LIN {X 0,Y 253.722,Z 799.815,A -85,B 0,C 180,E1 18671.44,E2 18671.44} C_VEL
LIN {X 0,Y 268.421,Z 770.688,A -85,B 0,C 180,E1 18677.162,E2 18677.162} C_VEL
LIN {X 0,Y 281.731,Z 738.919,A -85,B 0,C 180,E1 18681.257,E2 18681.257} C_VEL
LIN {X 0,Y 284.612,Z 730.237,A -85,B 0,C 180,E1 18682.199,E2 18682.199} C_VEL
LIN {X 0,Y 279.923,Z 708.728,A -85,B 0,C 180,E1 18687.264,E2 18687.264} C_VEL
LIN {X 0,Y 272.289,Z 686.779,A -85,B 0,C 180,E1 18693.595,E2 18693.595} C_VEL
LIN {X 0,Y 264.119,Z 669.28,A -85,B 0,C 180,E1 18700.544,E2 18700.544} C_VEL
LIN {X 0,Y 257.422,Z 656.995,A -85,B 0,C 180,E1 18708.127,E2 18708.127} C_VEL
LIN {X 0,Y 254.132,Z 650.458,A -85,B 0,C 180,E1 18714.879,E2 18714.879} C_VEL
LIN {X 0,Y 253.888,Z 650.396,A -85,B 0,C 180,E1 18725.138,E2 18725.138} C_VEL
LIN {X 0,Y 254.562,Z 652.061,A -85,B 0,C 180,E1 18727.374,E2 18727.374} C_VEL
LIN {X 0,Y 257.625,Z 657.599,A -85,B 0,C 180,E1 18733,E2 18733} C_VEL
LIN {X 0,Y 260.37,Z 676.439,A -85,B 0,C 180,E1 18739.556,E2 18739.556} C_VEL
LIN {X 0,Y 277.56,Z 705.99,A -85,B 0,C 180,E1 18753.063,E2 18753.063} C_VEL
LIN {X 0,Y 289.539,Z 719.07,A -85,B 0,C 180,E1 18759.84,E2 18759.84} C_VEL
LIN {X 0,Y 300.678,Z 730.907,A -85,B 0,C 180,E1 18766.755,E2 18766.755} C_VEL
LIN {X 0,Y 310.062,Z 741.061,A -85,B 0,C 180,E1 18773.393,E2 18773.393} C_VEL
LIN {X 0,Y 317.477,Z 748.305,A -85,B 0,C 180,E1 18779.146,E2 18779.146} C_VEL
LIN {X 0,Y 324.187,Z 754.391,A -85,B 0,C 180,E1 18785.145,E2 18785.145} C_VEL
LIN {X 0,Y 329.073,Z 760.266,A -85,B 0,C 180,E1 18791.212,E2 18791.212} C_VEL
LIN {X 0,Y 333.307,Z 763.024,A -85,B 0,C 180,E1 18796.872,E2 18796.872} C_VEL
LIN {X 0,Y 336.362,Z 764.049,A -85,B 0,C 180,E1 18802.239,E2 18802.239} C_VEL
LIN {X 0,Y 337.345,Z 765.358,A -85,B 0,C 180,E1 18807.428,E2 18807.428} C_VEL
LIN {X 0,Y 337.291,Z 765.495,A -85,B 0,C 180,E1 18812.573,E2 18812.573} C_VEL
LIN {X 0,Y 336.316,Z 764.064,A -85,B 0,C 180,E1 18817.923,E2 18817.923} C_VEL
LIN {X 0,Y 333.217,Z 763.056,A -85,B 0,C 180,E1 18823.132,E2 18823.132} C_VEL
LIN {X 0,Y 329.143,Z 760.264,A -85,B 0,C 180,E1 18828.784,E2 18828.784} C_VEL
LIN {X 0,Y 324.257,Z 754.4,A -85,B 0,C 180,E1 18834.85,E2 18834.85} C_VEL
LIN {X 0,Y 317.504,Z 748.261,A -85,B 0,C 180,E1 18840.862,E2 18840.862} C_VEL
LIN {X 0,Y 309.323,Z 739.929,A -85,B 0,C 180,E1 18847.257,E2 18847.257} C_VEL
LIN {X 0,Y 299.888,Z 729.733,A -85,B 0,C 180,E1 18853.843,E2 18853.843} C_VEL
LIN {X 0,Y 288.152,Z 717.936,A -85,B 0,C 180,E1 18860.906,E2 18860.906} C_VEL
LIN {X 0,Y 276.213,Z 704.369,A -85,B 0,C 180,E1 18867.689,E2 18867.689} C_VEL
LIN {X 0,Y 258.025,Z 670.823,A -85,B 0,C 180,E1 18883.393,E2 18883.393} C_VEL
LIN {X 0,Y 254.267,Z 663.867,A -85,B 0,C 180,E1 18888.836,E2 18888.836} C_VEL
LIN {X 0,Y 252.197,Z 658.099,A -85,B 0,C 180,E1 18894.827,E2 18894.827} C_VEL
LIN {X 0,Y 252.201,Z 658.014,A -85,B 0,C 180,E1 18904.297,E2 18904.297} C_VEL
LIN {X 0,Y 252.963,Z 660.074,A -85,B 0,C 180,E1 18906.977,E2 18906.977} C_VEL
LIN {X 0,Y 256.034,Z 666.467,A -85,B 0,C 180,E1 18912.914,E2 18912.914} C_VEL
LIN {X 0,Y 260.849,Z 675.753,A -85,B 0,C 180,E1 18918.61,E2 18918.61} C_VEL
LIN {X 0,Y 267.694,Z 691.294,A -85,B 0,C 180,E1 18925.184,E2 18925.184} C_VEL
LIN {X 0,Y 274.436,Z 712.152,A -85,B 0,C 180,E1 18931.6,E2 18931.6} C_VEL
LIN {X 0,Y 278.679,Z 732.602,A -85,B 0,C 180,E1 18936.691,E2 18936.691} C_VEL
LIN {X 0,Y 271.431,Z 751.922,A -85,B 0,C 180,E1 18938.973,E2 18938.973} C_VEL
LIN {X 0,Y 257.684,Z 781.058,A -85,B 0,C 180,E1 18943.356,E2 18943.356} C_VEL
LIN {X 0,Y 242.695,Z 808.411,A -85,B 0,C 180,E1 18949.666,E2 18949.666} C_VEL
LIN {X 0,Y 230.265,Z 829.686,A -85,B 0,C 180,E1 18957.149,E2 18957.149} C_VEL
LIN {X 0,Y 221.341,Z 845.658,A -85,B 0,C 180,E1 18965.769,E2 18965.769} C_VEL
LIN {X 0,Y 217.04,Z 855.186,A -85,B 0,C 180,E1 18973.797,E2 18973.797} C_VEL
LIN {X 0,Y 215.382,Z 860.762,A -85,B 0,C 180,E1 18981.918,E2 18981.918} C_VEL
LIN {X 0,Y 215.327,Z 862.605,A -85,B 0,C 180,E1 18990,E2 18990} C_VEL
LIN {X 0,Y 215.382,Z 860.762,A -85,B 0,C 180,E1 18998.082,E2 18998.082} C_VEL
LIN {X 0,Y 217.443,Z 854.155,A -85,B 0,C 180,E1 19007.213,E2 19007.213} C_VEL
LIN {X 0,Y 223.848,Z 841.066,A -85,B 0,C 180,E1 19017.165,E2 19017.165} C_VEL
LIN {X 0,Y 234.929,Z 821.817,A -85,B 0,C 180,E1 19025.991,E2 19025.991} C_VEL
LIN {X 0,Y 247.875,Z 799.283,A -85,B 0,C 180,E1 19032.747,E2 19032.747} C_VEL
LIN {X 0,Y 263.025,Z 770.451,A -85,B 0,C 180,E1 19038.445,E2 19038.445} C_VEL
LIN {X 0,Y 276.907,Z 738.464,A -85,B 0,C 180,E1 19042.564,E2 19042.564} C_VEL
LIN {X 0,Y 278.662,Z 732.639,A -85,B 0,C 180,E1 19043.306,E2 19043.306} C_VEL
LIN {X 0,Y 274.032,Z 710.65,A -85,B 0,C 180,E1 19048.811,E2 19048.811} C_VEL
LIN {X 0,Y 267.257,Z 690.159,A -85,B 0,C 180,E1 19055.22,E2 19055.22} C_VEL
LIN {X 0,Y 260.328,Z 674.883,A -85,B 0,C 180,E1 19061.9,E2 19061.9} C_VEL
LIN {X 0,Y 255.049,Z 664.367,A -85,B 0,C 180,E1 19068.666,E2 19068.666} C_VEL
LIN {X 0,Y 252.498,Z 658.186,A -85,B 0,C 180,E1 19074.846,E2 19074.846} C_VEL
LIN {X 0,Y 252.193,Z 658.115,A -85,B 0,C 180,E1 19085.173,E2 19085.173} C_VEL
LIN {X 0,Y 252.886,Z 661.098,A -85,B 0,C 180,E1 19088.181,E2 19088.181} C_VEL
LIN {X 0,Y 255.492,Z 666.126,A -85,B 0,C 180,E1 19093.172,E2 19093.172} C_VEL
LIN {X 0,Y 259.883,Z 675.45,A -85,B 0,C 180,E1 19099.011,E2 19099.011} C_VEL
LIN {X 0,Y 260.37,Z 676.439,A -85,B 0,C 180,E1 19099.556,E2 19099.556} C_VEL
LIN {X 0,Y 261.605,Z 683.787,A -85,B 0,C 180,E1 19101.921,E2 19101.921} C_VEL
LIN {X 0,Y 262.505,Z 696.627,A -85,B 0,C 180,E1 19105.243,E2 19105.243} C_VEL
LIN {X 0,Y 262.894,Z 697.628,A -85,B 0,C 180,E1 19105.664,E2 19105.664} C_VEL
LIN {X 0,Y 279.794,Z 719.558,A -85,B 0,C 180,E1 19116.535,E2 19116.535} C_VEL
LIN {X 0,Y 290.789,Z 731.877,A -85,B 0,C 180,E1 19123.202,E2 19123.202} C_VEL
LIN {X 0,Y 299.954,Z 741.66,A -85,B 0,C 180,E1 19129.218,E2 19129.218} C_VEL
LIN {X 0,Y 308.074,Z 750.087,A -85,B 0,C 180,E1 19135.117,E2 19135.117} C_VEL
LIN {X 0,Y 314.208,Z 756.261,A -85,B 0,C 180,E1 19140.159,E2 19140.159} C_VEL
LIN {X 0,Y 321.523,Z 762.613,A -85,B 0,C 180,E1 19146.889,E2 19146.889} C_VEL
LIN {X 0,Y 324.527,Z 766.633,A -85,B 0,C 180,E1 19150.939,E2 19150.939} C_VEL
LIN {X 0,Y 328.854,Z 769.575,A -85,B 0,C 180,E1 19156.691,E2 19156.691} C_VEL
LIN {X 0,Y 332,Z 770.682,A -85,B 0,C 180,E1 19162.137,E2 19162.137} C_VEL
LIN {X 0,Y 332.988,Z 771.949,A -85,B 0,C 180,E1 19167.394,E2 19167.394} C_VEL
LIN {X 0,Y 332.942,Z 772.067,A -85,B 0,C 180,E1 19172.606,E2 19172.606} C_VEL
LIN {X 0,Y 332.08,Z 770.689,A -85,B 0,C 180,E1 19177.861,E2 19177.861} C_VEL
LIN {X 0,Y 328.094,Z 769.257,A -85,B 0,C 180,E1 19184.273,E2 19184.273} C_VEL
LIN {X 0,Y 323.429,Z 765.318,A -85,B 0,C 180,E1 19190.561,E2 19190.561} C_VEL
LIN {X 0,Y 319.061,Z 760.427,A -85,B 0,C 180,E1 19195.622,E2 19195.622} C_VEL
LIN {X 0,Y 311.602,Z 753.026,A -85,B 0,C 180,E1 19202.309,E2 19202.309} C_VEL
LIN {X 0,Y 303.516,Z 744.804,A -85,B 0,C 180,E1 19208.443,E2 19208.443} C_VEL
LIN {X 0,Y 293.878,Z 734.884,A -85,B 0,C 180,E1 19214.917,E2 19214.917} C_VEL
LIN {X 0,Y 283.124,Z 723.825,A -85,B 0,C 180,E1 19221.367,E2 19221.367} C_VEL
LIN {X 0,Y 270.484,Z 709.163,A -85,B 0,C 180,E1 19228.722,E2 19228.722} C_VEL
LIN {X 0,Y 255.071,Z 677.938,A -85,B 0,C 180,E1 19243.844,E2 19243.844} C_VEL
LIN {X 0,Y 251.743,Z 671.095,A -85,B 0,C 180,E1 19249.38,E2 19249.38} C_VEL
LIN {X 0,Y 250.18,Z 665.733,A -85,B 0,C 180,E1 19254.786,E2 19254.786} C_VEL
LIN {X 0,Y 250.491,Z 665.82,A -85,B 0,C 180,E1 19265.195,E2 19265.195} C_VEL
LIN {X 0,Y 253.676,Z 674.085,A -85,B 0,C 180,E1 19272.707,E2 19272.707} C_VEL
LIN {X 0,Y 258.959,Z 685.721,A -85,B 0,C 180,E1 19279.637,E2 19279.637} C_VEL
LIN {X 0,Y 265.288,Z 702.329,A -85,B 0,C 180,E1 19286.29,E2 19286.29} C_VEL
LIN {X 0,Y 270.915,Z 723.903,A -85,B 0,C 180,E1 19292.736,E2 19292.736} C_VEL
LIN {X 0,Y 272.755,Z 736.639,A -85,B 0,C 180,E1 19295.931,E2 19295.931} C_VEL
LIN {X 0,Y 258.291,Z 769.097,A -85,B 0,C 180,E1 19300.031,E2 19300.031} C_VEL
LIN {X 0,Y 243.885,Z 795.806,A -85,B 0,C 180,E1 19305.191,E2 19305.191} C_VEL
LIN {X 0,Y 229.737,Z 819.508,A -85,B 0,C 180,E1 19312.022,E2 19312.022} C_VEL
LIN {X 0,Y 217.666,Z 839.049,A -85,B 0,C 180,E1 19320.862,E2 19320.862} C_VEL
LIN {X 0,Y 210.689,Z 851.849,A -85,B 0,C 180,E1 19330.041,E2 19330.041} C_VEL
LIN {X 0,Y 207.856,Z 859.051,A -85,B 0,C 180,E1 19338.863,E2 19338.863} C_VEL
LIN {X 0,Y 207.251,Z 861.906,A -85,B 0,C 180,E1 19345.811,E2 19345.811} C_VEL
LIN {X 0,Y 207.435,Z 862.372,A -85,B 0,C 180,E1 19350,E2 19350} C_VEL
LIN {X 0,Y 207.523,Z 860.527,A -85,B 0,C 180,E1 19358.39,E2 19358.39} C_VEL
LIN {X 0,Y 209.752,Z 853.917,A -85,B 0,C 180,E1 19367.865,E2 19367.865} C_VEL
LIN {X 0,Y 216.67,Z 840.826,A -85,B 0,C 180,E1 19378.143,E2 19378.143} C_VEL
LIN {X 0,Y 227.715,Z 822.692,A -85,B 0,C 180,E1 19386.755,E2 19386.755} C_VEL
LIN {X 0,Y 241.164,Z 800.565,A -85,B 0,C 180,E1 19393.677,E2 19393.677} C_VEL
LIN {X 0,Y 256.69,Z 772.229,A -85,B 0,C 180,E1 19399.447,E2 19399.447} C_VEL
LIN {X 0,Y 270.793,Z 741.417,A -85,B 0,C 180,E1 19403.578,E2 19403.578} C_VEL
LIN {X 0,Y 272.727,Z 736.789,A -85,B 0,C 180,E1 19404.045,E2 19404.045} C_VEL
LIN {X 0,Y 269.429,Z 717.127,A -85,B 0,C 180,E1 19409.153,E2 19409.153} C_VEL
LIN {X 0,Y 263.704,Z 697.585,A -85,B 0,C 180,E1 19415.348,E2 19415.348} C_VEL
LIN {X 0,Y 257.508,Z 682.395,A -85,B 0,C 180,E1 19422.027,E2 19422.027} C_VEL
LIN {X 0,Y 252.531,Z 671.634,A -85,B 0,C 180,E1 19429.208,E2 19429.208} C_VEL
LIN {X 0,Y 250.197,Z 665.645,A -85,B 0,C 180,E1 19435.668,E2 19435.668} C_VEL
LIN {X 0,Y 250.394,Z 665.875,A -85,B 0,C 180,E1 19445.863,E2 19445.863} C_VEL
LIN {X 0,Y 253.009,Z 673.709,A -85,B 0,C 180,E1 19452.974,E2 19452.974} C_VEL
LIN {X 0,Y 257.04,Z 683.169,A -85,B 0,C 180,E1 19458.987,E2 19458.987} C_VEL
LIN {X 0,Y 262.894,Z 697.628,A -85,B 0,C 180,E1 19465.664,E2 19465.664} C_VEL
LIN {X 0,Y 264.943,Z 707.476,A -85,B 0,C 180,E1 19468.776,E2 19468.776} C_VEL
LIN {X 0,Y 267.331,Z 717.144,A -85,B 0,C 180,E1 19471.876,E2 19471.876} C_VEL
LIN {X 0,Y 280.458,Z 731.903,A -85,B 0,C 180,E1 19479.567,E2 19479.567} C_VEL
LIN {X 0,Y 291.702,Z 743.909,A -85,B 0,C 180,E1 19486.612,E2 19486.612} C_VEL
LIN {X 0,Y 301.367,Z 754.364,A -85,B 0,C 180,E1 19493.503,E2 19493.503} C_VEL
LIN {X 0,Y 309.025,Z 761.994,A -85,B 0,C 180,E1 19499.606,E2 19499.606} C_VEL
LIN {X 0,Y 315.782,Z 767.906,A -85,B 0,C 180,E1 19505.648,E2 19505.648} C_VEL
LIN {X 0,Y 320.017,Z 773.144,A -85,B 0,C 180,E1 19511.135,E2 19511.135} C_VEL
LIN {X 0,Y 325.063,Z 776.401,A -85,B 0,C 180,E1 19518.006,E2 19518.006} C_VEL
LIN {X 0,Y 327.313,Z 777.086,A -85,B 0,C 180,E1 19522.023,E2 19522.023} C_VEL
LIN {X 0,Y 328.378,Z 778.338,A -85,B 0,C 180,E1 19527.357,E2 19527.357} C_VEL
LIN {X 0,Y 328.321,Z 778.457,A -85,B 0,C 180,E1 19532.643,E2 19532.643} C_VEL
LIN {X 0,Y 327.409,Z 777.086,A -85,B 0,C 180,E1 19537.974,E2 19537.974} C_VEL
LIN {X 0,Y 324.034,Z 775.932,A -85,B 0,C 180,E1 19543.511,E2 19543.511} C_VEL
LIN {X 0,Y 319.707,Z 772.73,A -85,B 0,C 180,E1 19549.36,E2 19549.36} C_VEL
LIN {X 0,Y 315.812,Z 767.886,A -85,B 0,C 180,E1 19554.364,E2 19554.364} C_VEL
LIN {X 0,Y 309.067,Z 761.952,A -85,B 0,C 180,E1 19560.4,E2 19560.4} C_VEL
LIN {X 0,Y 301.418,Z 754.31,A -85,B 0,C 180,E1 19566.51,E2 19566.51} C_VEL
LIN {X 0,Y 291.708,Z 743.862,A -85,B 0,C 180,E1 19573.389,E2 19573.389} C_VEL
LIN {X 0,Y 280.275,Z 731.939,A -85,B 0,C 180,E1 19580.485,E2 19580.485} C_VEL
LIN {X 0,Y 267.117,Z 716.998,A -85,B 0,C 180,E1 19588.236,E2 19588.236} C_VEL
LIN {X 0,Y 252.216,Z 685.865,A -85,B 0,C 180,E1 19603.839,E2 19603.839} C_VEL
LIN {X 0,Y 249.209,Z 678.563,A -85,B 0,C 180,E1 19609.492,E2 19609.492} C_VEL
LIN {X 0,Y 247.798,Z 673.138,A -85,B 0,C 180,E1 19615.614,E2 19615.614} C_VEL
LIN {X 0,Y 248.364,Z 673.568,A -85,B 0,C 180,E1 19625.24,E2 19625.24} C_VEL
LIN {X 0,Y 251.754,Z 683.542,A -85,B 0,C 180,E1 19633.913,E2 19633.913} C_VEL
LIN {X 0,Y 256.791,Z 695.706,A -85,B 0,C 180,E1 19640.71,E2 19640.71} C_VEL
LIN {X 0,Y 262.017,Z 712.293,A -85,B 0,C 180,E1 19647.06,E2 19647.06} C_VEL
LIN {X 0,Y 266.396,Z 733.834,A -85,B 0,C 180,E1 19653.416,E2 19653.416} C_VEL
LIN {X 0,Y 266.903,Z 738.98,A -85,B 0,C 180,E1 19654.767,E2 19654.767} C_VEL
LIN {X 0,Y 252.624,Z 769.975,A -85,B 0,C 180,E1 19658.819,E2 19658.819} C_VEL
LIN {X 0,Y 236.375,Z 798.637,A -85,B 0,C 180,E1 19664.554,E2 19664.554} C_VEL
LIN {X 0,Y 222.467,Z 820.638,A -85,B 0,C 180,E1 19671.272,E2 19671.272} C_VEL
LIN {X 0,Y 209.559,Z 840.587,A -85,B 0,C 180,E1 19680.812,E2 19680.812} C_VEL
LIN {X 0,Y 202.08,Z 853.678,A -85,B 0,C 180,E1 19691.432,E2 19691.432} C_VEL
LIN {X 0,Y 199.638,Z 860.292,A -85,B 0,C 180,E1 19701.276,E2 19701.276} C_VEL
LIN {X 0,Y 199.53,Z 862.139,A -85,B 0,C 180,E1 19710,E2 19710} C_VEL
LIN {X 0,Y 199.756,Z 859.695,A -85,B 0,C 180,E1 19719.884,E2 19719.884} C_VEL
LIN {X 0,Y 203.144,Z 851.611,A -85,B 0,C 180,E1 19730.734,E2 19730.734} C_VEL
LIN {X 0,Y 211.073,Z 838.099,A -85,B 0,C 180,E1 19740.615,E2 19740.615} C_VEL
LIN {X 0,Y 223.564,Z 819.097,A -85,B 0,C 180,E1 19749.311,E2 19749.311} C_VEL
LIN {X 0,Y 239.452,Z 793.571,A -85,B 0,C 180,E1 19756.648,E2 19756.648} C_VEL
LIN {X 0,Y 254.977,Z 765.277,A -85,B 0,C 180,E1 19761.886,E2 19761.886} C_VEL
LIN {X 0,Y 266.857,Z 739.017,A -85,B 0,C 180,E1 19765.239,E2 19765.239} C_VEL
LIN {X 0,Y 263.637,Z 718.627,A -85,B 0,C 180,E1 19770.942,E2 19770.942} C_VEL
LIN {X 0,Y 258.413,Z 700.308,A -85,B 0,C 180,E1 19777.33,E2 19777.33} C_VEL
LIN {X 0,Y 252.837,Z 685.749,A -85,B 0,C 180,E1 19784.544,E2 19784.544} C_VEL
LIN {X 0,Y 249.919,Z 678.958,A -85,B 0,C 180,E1 19789.535,E2 19789.535} C_VEL
LIN {X 0,Y 248.104,Z 673.261,A -85,B 0,C 180,E1 19795.632,E2 19795.632} C_VEL
LIN {X 0,Y 248.023,Z 673.333,A -85,B 0,C 180,E1 19805.26,E2 19805.26} C_VEL
LIN {X 0,Y 250.283,Z 681.386,A -85,B 0,C 180,E1 19812.895,E2 19812.895} C_VEL
LIN {X 0,Y 253.863,Z 690.817,A -85,B 0,C 180,E1 19818.929,E2 19818.929} C_VEL
LIN {X 0,Y 267.331,Z 717.144,A -85,B 0,C 180,E1 19831.876,E2 19831.876} C_VEL
LIN {X 0,Y 270.192,Z 726.565,A -85,B 0,C 180,E1 19834.981,E2 19834.981} C_VEL
LIN {X 0,Y 273.227,Z 735.611,A -85,B 0,C 180,E1 19838.092,E2 19838.092} C_VEL
LIN {X 0,Y 282.991,Z 746.158,A -85,B 0,C 180,E1 19844.074,E2 19844.074} C_VEL
LIN {X 0,Y 293.02,Z 756.622,A -85,B 0,C 180,E1 19850.816,E2 19850.816} C_VEL
LIN {X 0,Y 301.566,Z 765.232,A -85,B 0,C 180,E1 19857.259,E2 19857.259} C_VEL
LIN {X 0,Y 308.855,Z 772.625,A -85,B 0,C 180,E1 19863.82,E2 19863.82} C_VEL
LIN {X 0,Y 313.225,Z 776.998,A -85,B 0,C 180,E1 19868.506,E2 19868.506} C_VEL
LIN {X 0,Y 316.801,Z 780.734,A -85,B 0,C 180,E1 19873.336,E2 19873.336} C_VEL
LIN {X 0,Y 320.85,Z 782.844,A -85,B 0,C 180,E1 19879.12,E2 19879.12} C_VEL
LIN {X 0,Y 322.381,Z 783.297,A -85,B 0,C 180,E1 19881.9,E2 19881.9} C_VEL
LIN {X 0,Y 323.527,Z 784.547,A -85,B 0,C 180,E1 19887.318,E2 19887.318} C_VEL
LIN {X 0,Y 323.456,Z 784.667,A -85,B 0,C 180,E1 19892.683,E2 19892.683} C_VEL
LIN {X 0,Y 322.467,Z 783.31,A -85,B 0,C 180,E1 19898.097,E2 19898.097} C_VEL
LIN {X 0,Y 318.976,Z 782.056,A -85,B 0,C 180,E1 19903.729,E2 19903.729} C_VEL
LIN {X 0,Y 314.537,Z 778.63,A -85,B 0,C 180,E1 19909.691,E2 19909.691} C_VEL
LIN {X 0,Y 310.465,Z 773.757,A -85,B 0,C 180,E1 19914.812,E2 19914.812} C_VEL
LIN {X 0,Y 302.785,Z 766.382,A -85,B 0,C 180,E1 19921.774,E2 19921.774} C_VEL
LIN {X 0,Y 294.608,Z 758.134,A -85,B 0,C 180,E1 19928.076,E2 19928.076} C_VEL
LIN {X 0,Y 284.689,Z 747.712,A -85,B 0,C 180,E1 19934.89,E2 19934.89} C_VEL
LIN {X 0,Y 273.756,Z 736.522,A -85,B 0,C 180,E1 19941.517,E2 19941.517} C_VEL
LIN {X 0,Y 254.357,Z 710.118,A -85,B 0,C 180,E1 19955.37,E2 19955.37} C_VEL
LIN {X 0,Y 249.142,Z 693.874,A -85,B 0,C 180,E1 19963.634,E2 19963.634} C_VEL
LIN {X 0,Y 246.628,Z 686.171,A -85,B 0,C 180,E1 19969.381,E2 19969.381} C_VEL
LIN {X 0,Y 245.453,Z 681.076,A -85,B 0,C 180,E1 19974.685,E2 19974.685} C_VEL
LIN {X 0,Y 245.4,Z 680.546,A -85,B 0,C 180,E1 19983.531,E2 19983.531} C_VEL
LIN {X 0,Y 247.876,Z 687.96,A -85,B 0,C 180,E1 19991.643,E2 19991.643} C_VEL
LIN {X 0,Y 252.355,Z 700.365,A -85,B 0,C 180,E1 19999.26,E2 19999.26} C_VEL
LIN {X 0,Y 256.943,Z 716.004,A -85,B 0,C 180,E1 20005.726,E2 20005.726} C_VEL
LIN {X 0,Y 260.602,Z 736.458,A -85,B 0,C 180,E1 20012.176,E2 20012.176} C_VEL
LIN {X 0,Y 260.662,Z 743.169,A -85,B 0,C 180,E1 20013.835,E2 20013.835} C_VEL
LIN {X 0,Y 245.083,Z 774.319,A -85,B 0,C 180,E1 20018.144,E2 20018.144} C_VEL
LIN {X 0,Y 228.716,Z 801.714,A -85,B 0,C 180,E1 20023.968,E2 20023.968} C_VEL
LIN {X 0,Y 212.983,Z 825.107,A -85,B 0,C 180,E1 20031.835,E2 20031.835} C_VEL
LIN {X 0,Y 201.451,Z 841.893,A -85,B 0,C 180,E1 20040.756,E2 20040.756} C_VEL
LIN {X 0,Y 193.97,Z 854.473,A -85,B 0,C 180,E1 20051.807,E2 20051.807} C_VEL
LIN {X 0,Y 191.776,Z 860.056,A -85,B 0,C 180,E1 20060.915,E2 20060.915} C_VEL
LIN {X 0,Y 191.639,Z 861.906,A -85,B 0,C 180,E1 20070,E2 20070} C_VEL
LIN {X 0,Y 191.891,Z 859.459,A -85,B 0,C 180,E1 20080.293,E2 20080.293} C_VEL
LIN {X 0,Y 194.832,Z 852.761,A -85,B 0,C 180,E1 20090.063,E2 20090.063} C_VEL
LIN {X 0,Y 202.511,Z 840.347,A -85,B 0,C 180,E1 20100.309,E2 20100.309} C_VEL
LIN {X 0,Y 215.803,Z 821.038,A -85,B 0,C 180,E1 20109.807,E2 20109.807} C_VEL
LIN {X 0,Y 230.799,Z 798.399,A -85,B 0,C 180,E1 20116.87,E2 20116.87} C_VEL
LIN {X 0,Y 247.71,Z 769.74,A -85,B 0,C 180,E1 20122.616,E2 20122.616} C_VEL
LIN {X 0,Y 261.064,Z 741.913,A -85,B 0,C 180,E1 20126.339,E2 20126.339} C_VEL
LIN {X 0,Y 258.358,Z 722.534,A -85,B 0,C 180,E1 20132.05,E2 20132.05} C_VEL
LIN {X 0,Y 254.221,Z 705.988,A -85,B 0,C 180,E1 20138.154,E2 20138.154} C_VEL
LIN {X 0,Y 249.528,Z 692.442,A -85,B 0,C 180,E1 20145.149,E2 20145.149} C_VEL
LIN {X 0,Y 246.338,Z 684.839,A -85,B 0,C 180,E1 20151.588,E2 20151.588} C_VEL
LIN {X 0,Y 245.382,Z 680.6,A -85,B 0,C 180,E1 20156.469,E2 20156.469} C_VEL
LIN {X 0,Y 245.44,Z 681.115,A -85,B 0,C 180,E1 20165.315,E2 20165.315} C_VEL
LIN {X 0,Y 247.516,Z 689.416,A -85,B 0,C 180,E1 20173.177,E2 20173.177} C_VEL
LIN {X 0,Y 251.341,Z 701.047,A -85,B 0,C 180,E1 20180.272,E2 20180.272} C_VEL
LIN {X 0,Y 266.088,Z 727.988,A -85,B 0,C 180,E1 20193.995,E2 20193.995} C_VEL
LIN {X 0,Y 273.227,Z 735.611,A -85,B 0,C 180,E1 20198.092,E2 20198.092} C_VEL
LIN {X 0,Y 275.088,Z 739.562,A -85,B 0,C 180,E1 20199.679,E2 20199.679} C_VEL
LIN {X 0,Y 277.859,Z 751.96,A -85,B 0,C 180,E1 20203.965,E2 20203.965} C_VEL
LIN {X 0,Y 278.458,Z 752.663,A -85,B 0,C 180,E1 20204.376,E2 20204.376} C_VEL
LIN {X 0,Y 288.059,Z 762.798,A -85,B 0,C 180,E1 20210.896,E2 20210.896} C_VEL
LIN {X 0,Y 296.642,Z 771.433,A -85,B 0,C 180,E1 20217.399,E2 20217.399} C_VEL
LIN {X 0,Y 303.728,Z 778.633,A -85,B 0,C 180,E1 20223.81,E2 20223.81} C_VEL
LIN {X 0,Y 308.361,Z 783.367,A -85,B 0,C 180,E1 20228.9,E2 20228.9} C_VEL
LIN {X 0,Y 313.083,Z 787.623,A -85,B 0,C 180,E1 20235.294,E2 20235.294} C_VEL
LIN {X 0,Y 317.191,Z 789.318,A -85,B 0,C 180,E1 20241.767,E2 20241.767} C_VEL
LIN {X 0,Y 318.431,Z 790.546,A -85,B 0,C 180,E1 20247.275,E2 20247.275} C_VEL
LIN {X 0,Y 318.345,Z 790.669,A -85,B 0,C 180,E1 20252.795,E2 20252.795} C_VEL
LIN {X 0,Y 317.288,Z 789.321,A -85,B 0,C 180,E1 20258.23,E2 20258.23} C_VEL
LIN {X 0,Y 313.056,Z 787.646,A -85,B 0,C 180,E1 20264.688,E2 20264.688} C_VEL
LIN {X 0,Y 308.342,Z 783.344,A -85,B 0,C 180,E1 20271.091,E2 20271.091} C_VEL
LIN {X 0,Y 303.159,Z 778.157,A -85,B 0,C 180,E1 20276.711,E2 20276.711} C_VEL
LIN {X 0,Y 296.673,Z 771.442,A -85,B 0,C 180,E1 20282.583,E2 20282.583} C_VEL
LIN {X 0,Y 288.152,Z 762.747,A -85,B 0,C 180,E1 20289.089,E2 20289.089} C_VEL
LIN {X 0,Y 279.195,Z 753.379,A -85,B 0,C 180,E1 20295.166,E2 20295.166} C_VEL
LIN {X 0,Y 268.531,Z 742.392,A -85,B 0,C 180,E1 20301.663,E2 20301.663} C_VEL
LIN {X 0,Y 249.27,Z 714.051,A -85,B 0,C 180,E1 20316.938,E2 20316.938} C_VEL
LIN {X 0,Y 245.354,Z 699.556,A -85,B 0,C 180,E1 20324.79,E2 20324.79} C_VEL
LIN {X 0,Y 243.705,Z 693.637,A -85,B 0,C 180,E1 20329.252,E2 20329.252} C_VEL
LIN {X 0,Y 242.537,Z 687.968,A -85,B 0,C 180,E1 20336.415,E2 20336.415} C_VEL
LIN {X 0,Y 242.982,Z 688.49,A -85,B 0,C 180,E1 20344.453,E2 20344.453} C_VEL
LIN {X 0,Y 245.319,Z 697.232,A -85,B 0,C 180,E1 20352.874,E2 20352.874} C_VEL
LIN {X 0,Y 249.004,Z 708.381,A -85,B 0,C 180,E1 20359.53,E2 20359.53} C_VEL
LIN {X 0,Y 252.723,Z 724.279,A -85,B 0,C 180,E1 20366.02,E2 20366.02} C_VEL
LIN {X 0,Y 255.317,Z 743.846,A -85,B 0,C 180,E1 20372.248,E2 20372.248} C_VEL
LIN {X 0,Y 253.134,Z 749.625,A -85,B 0,C 180,E1 20373.136,E2 20373.136} C_VEL
LIN {X 0,Y 236.94,Z 779.822,A -85,B 0,C 180,E1 20377.637,E2 20377.637} C_VEL
LIN {X 0,Y 219.641,Z 806.646,A -85,B 0,C 180,E1 20383.959,E2 20383.959} C_VEL
LIN {X 0,Y 204.93,Z 827.3,A -85,B 0,C 180,E1 20391.513,E2 20391.513} C_VEL
LIN {X 0,Y 192.279,Z 844.701,A -85,B 0,C 180,E1 20401.806,E2 20401.806} C_VEL
LIN {X 0,Y 186.354,Z 854.235,A -85,B 0,C 180,E1 20411.035,E2 20411.035} C_VEL
LIN {X 0,Y 183.812,Z 860.045,A -85,B 0,C 180,E1 20421.206,E2 20421.206} C_VEL
LIN {X 0,Y 183.732,Z 861.672,A -85,B 0,C 180,E1 20430,E2 20430} C_VEL
LIN {X 0,Y 183.905,Z 859.821,A -85,B 0,C 180,E1 20439.477,E2 20439.477} C_VEL
LIN {X 0,Y 187.185,Z 852.693,A -85,B 0,C 180,E1 20450.716,E2 20450.716} C_VEL
LIN {X 0,Y 195.871,Z 839.668,A -85,B 0,C 180,E1 20461.777,E2 20461.777} C_VEL
LIN {X 0,Y 210.503,Z 819.621,A -85,B 0,C 180,E1 20471.706,E2 20471.706} C_VEL
LIN {X 0,Y 226.446,Z 796.471,A -85,B 0,C 180,E1 20478.781,E2 20478.781} C_VEL
LIN {X 0,Y 243.513,Z 768.385,A -85,B 0,C 180,E1 20484.308,E2 20484.308} C_VEL
LIN {X 0,Y 255.183,Z 745.396,A -85,B 0,C 180,E1 20487.382,E2 20487.382} C_VEL
LIN {X 0,Y 253.309,Z 727.382,A -85,B 0,C 180,E1 20492.896,E2 20492.896} C_VEL
LIN {X 0,Y 250.046,Z 712.218,A -85,B 0,C 180,E1 20498.704,E2 20498.704} C_VEL
LIN {X 0,Y 246.045,Z 699.068,A -85,B 0,C 180,E1 20505.758,E2 20505.758} C_VEL
LIN {X 0,Y 243.565,Z 692.383,A -85,B 0,C 180,E1 20511.491,E2 20511.491} C_VEL
LIN {X 0,Y 242.829,Z 688.092,A -85,B 0,C 180,E1 20516.432,E2 20516.432} C_VEL
LIN {X 0,Y 242.534,Z 687.975,A -85,B 0,C 180,E1 20523.585,E2 20523.585} C_VEL
LIN {X 0,Y 243.824,Z 694.262,A -85,B 0,C 180,E1 20531.232,E2 20531.232} C_VEL
LIN {X 0,Y 246.886,Z 705.707,A -85,B 0,C 180,E1 20538.788,E2 20538.788} C_VEL
LIN {X 0,Y 259.387,Z 731.945,A -85,B 0,C 180,E1 20552.684,E2 20552.684} C_VEL
LIN {X 0,Y 272.578,Z 746.104,A -85,B 0,C 180,E1 20560.607,E2 20560.607} C_VEL
LIN {X 0,Y 278.458,Z 752.663,A -85,B 0,C 180,E1 20564.376,E2 20564.376} C_VEL
LIN {X 0,Y 280.576,Z 758.322,A -85,B 0,C 180,E1 20566.758,E2 20566.758} C_VEL
LIN {X 0,Y 281.99,Z 767.756,A -85,B 0,C 180,E1 20570.319,E2 20570.319} C_VEL
LIN {X 0,Y 282.475,Z 768.418,A -85,B 0,C 180,E1 20570.735,E2 20570.735} C_VEL
LIN {X 0,Y 291.673,Z 777.651,A -85,B 0,C 180,E1 20577.768,E2 20577.768} C_VEL
LIN {X 0,Y 299.092,Z 784.967,A -85,B 0,C 180,E1 20584.472,E2 20584.472} C_VEL
LIN {X 0,Y 304.425,Z 790.85,A -85,B 0,C 180,E1 20590.911,E2 20590.911} C_VEL
LIN {X 0,Y 309.585,Z 794.357,A -85,B 0,C 180,E1 20598.005,E2 20598.005} C_VEL
LIN {X 0,Y 311.718,Z 795.096,A -85,B 0,C 180,E1 20601.621,E2 20601.621} C_VEL
LIN {X 0,Y 312.988,Z 796.275,A -85,B 0,C 180,E1 20607.227,E2 20607.227} C_VEL
LIN {X 0,Y 312.924,Z 796.374,A -85,B 0,C 180,E1 20612.773,E2 20612.773} C_VEL
LIN {X 0,Y 311.815,Z 795.098,A -85,B 0,C 180,E1 20618.376,E2 20618.376} C_VEL
LIN {X 0,Y 307.959,Z 793.556,A -85,B 0,C 180,E1 20624.23,E2 20624.23} C_VEL
LIN {X 0,Y 302.608,Z 788.701,A -85,B 0,C 180,E1 20631.511,E2 20631.511} C_VEL
LIN {X 0,Y 298.111,Z 784.16,A -85,B 0,C 180,E1 20636.417,E2 20636.417} C_VEL
LIN {X 0,Y 290.232,Z 776.258,A -85,B 0,C 180,E1 20643.412,E2 20643.412} C_VEL
LIN {X 0,Y 281.128,Z 766.963,A -85,B 0,C 180,E1 20650.261,E2 20650.261} C_VEL
LIN {X 0,Y 271.197,Z 756.653,A -85,B 0,C 180,E1 20656.845,E2 20656.845} C_VEL
LIN {X 0,Y 259.205,Z 743.472,A -85,B 0,C 180,E1 20664.254,E2 20664.254} C_VEL
LIN {X 0,Y 243.941,Z 717.412,A -85,B 0,C 180,E1 20678.989,E2 20678.989} C_VEL
LIN {X 0,Y 241.59,Z 705.953,A -85,B 0,C 180,E1 20685.476,E2 20685.476} C_VEL
LIN {X 0,Y 239.671,Z 698.252,A -85,B 0,C 180,E1 20692.735,E2 20692.735} C_VEL
LIN {X 0,Y 239.578,Z 695.336,A -85,B 0,C 180,E1 20696.37,E2 20696.37} C_VEL
LIN {X 0,Y 239.892,Z 695.423,A -85,B 0,C 180,E1 20703.612,E2 20703.612} C_VEL
LIN {X 0,Y 242.02,Z 704.358,A -85,B 0,C 180,E1 20712.641,E2 20712.641} C_VEL
LIN {X 0,Y 245.267,Z 716.056,A -85,B 0,C 180,E1 20719.608,E2 20719.608} C_VEL
LIN {X 0,Y 248.369,Z 732.945,A -85,B 0,C 180,E1 20726.511,E2 20726.511} C_VEL
LIN {X 0,Y 249.537,Z 748.03,A -85,B 0,C 180,E1 20731.431,E2 20731.431} C_VEL
LIN {X 0,Y 232.183,Z 779.482,A -85,B 0,C 180,E1 20736.048,E2 20736.048} C_VEL
LIN {X 0,Y 214.347,Z 806.08,A -85,B 0,C 180,E1 20742.308,E2 20742.308} C_VEL
LIN {X 0,Y 199.123,Z 826.466,A -85,B 0,C 180,E1 20749.767,E2 20749.767} C_VEL
LIN {X 0,Y 185.192,Z 844.462,A -85,B 0,C 180,E1 20760.624,E2 20760.624} C_VEL
LIN {X 0,Y 177.75,Z 855.67,A -85,B 0,C 180,E1 20772.655,E2 20772.655} C_VEL
LIN {X 0,Y 176.032,Z 859.585,A -85,B 0,C 180,E1 20780.095,E2 20780.095} C_VEL
LIN {X 0,Y 175.824,Z 861.438,A -85,B 0,C 180,E1 20790,E2 20790} C_VEL
LIN {X 0,Y 176.032,Z 859.585,A -85,B 0,C 180,E1 20799.905,E2 20799.905} C_VEL
LIN {X 0,Y 179.387,Z 852.915,A -85,B 0,C 180,E1 20811.083,E2 20811.083} C_VEL
LIN {X 0,Y 188.63,Z 839.986,A -85,B 0,C 180,E1 20822.71,E2 20822.71} C_VEL
LIN {X 0,Y 203.602,Z 820.558,A -85,B 0,C 180,E1 20832.732,E2 20832.732} C_VEL
LIN {X 0,Y 220.092,Z 797.923,A -85,B 0,C 180,E1 20839.935,E2 20839.935} C_VEL
LIN {X 0,Y 238.271,Z 769.263,A -85,B 0,C 180,E1 20845.697,E2 20845.697} C_VEL
LIN {X 0,Y 249.336,Z 748.35,A -85,B 0,C 180,E1 20848.545,E2 20848.545} C_VEL
LIN {X 0,Y 248.168,Z 731.301,A -85,B 0,C 180,E1 20854.09,E2 20854.09} C_VEL
LIN {X 0,Y 245.282,Z 716.057,A -85,B 0,C 180,E1 20860.382,E2 20860.382} C_VEL
LIN {X 0,Y 242.03,Z 704.336,A -85,B 0,C 180,E1 20867.36,E2 20867.36} C_VEL
LIN {X 0,Y 239.873,Z 695.468,A -85,B 0,C 180,E1 20876.388,E2 20876.388} C_VEL
LIN {X 0,Y 239.571,Z 695.353,A -85,B 0,C 180,E1 20883.63,E2 20883.63} C_VEL
LIN {X 0,Y 240.938,Z 703.7,A -85,B 0,C 180,E1 20892.712,E2 20892.712} C_VEL
LIN {X 0,Y 243.224,Z 713.593,A -85,B 0,C 180,E1 20899.082,E2 20899.082} C_VEL
LIN {X 0,Y 255.644,Z 739.617,A -85,B 0,C 180,E1 20913.477,E2 20913.477} C_VEL
LIN {X 0,Y 268.609,Z 753.688,A -85,B 0,C 180,E1 20921.482,E2 20921.482} C_VEL
LIN {X 0,Y 277.654,Z 763.501,A -85,B 0,C 180,E1 20927.411,E2 20927.411} C_VEL
LIN {X 0,Y 282.475,Z 768.418,A -85,B 0,C 180,E1 20930.735,E2 20930.735} C_VEL
LIN {X 0,Y 284.075,Z 773.582,A -85,B 0,C 180,E1 20933.155,E2 20933.155} C_VEL
LIN {X 0,Y 284.91,Z 781.962,A -85,B 0,C 180,E1 20936.776,E2 20936.776} C_VEL
LIN {X 0,Y 285.339,Z 782.522,A -85,B 0,C 180,E1 20937.194,E2 20937.194} C_VEL
LIN {X 0,Y 292.106,Z 789.493,A -85,B 0,C 180,E1 20943.276,E2 20943.276} C_VEL
LIN {X 0,Y 297.4,Z 794.816,A -85,B 0,C 180,E1 20949.123,E2 20949.123} C_VEL
LIN {X 0,Y 302.175,Z 798.931,A -85,B 0,C 180,E1 20955.491,E2 20955.491} C_VEL
LIN {X 0,Y 306.062,Z 800.589,A -85,B 0,C 180,E1 20961.661,E2 20961.661} C_VEL
LIN {X 0,Y 307.338,Z 801.767,A -85,B 0,C 180,E1 20967.176,E2 20967.176} C_VEL
LIN {X 0,Y 307.259,Z 801.872,A -85,B 0,C 180,E1 20972.824,E2 20972.824} C_VEL
LIN {X 0,Y 306.037,Z 800.592,A -85,B 0,C 180,E1 20978.535,E2 20978.535} C_VEL
LIN {X 0,Y 302.078,Z 798.941,A -85,B 0,C 180,E1 20984.513,E2 20984.513} C_VEL
LIN {X 0,Y 297.443,Z 794.829,A -85,B 0,C 180,E1 20990.874,E2 20990.874} C_VEL
LIN {X 0,Y 292.113,Z 789.412,A -85,B 0,C 180,E1 20996.739,E2 20996.739} C_VEL
LIN {X 0,Y 285.174,Z 782.326,A -85,B 0,C 180,E1 21002.956,E2 21002.956} C_VEL
LIN {X 0,Y 276.12,Z 773.087,A -85,B 0,C 180,E1 21009.849,E2 21009.849} C_VEL
LIN {X 0,Y 265.652,Z 762.279,A -85,B 0,C 180,E1 21016.843,E2 21016.843} C_VEL
LIN {X 0,Y 252.916,Z 748.346,A -85,B 0,C 180,E1 21024.886,E2 21024.886} C_VEL
LIN {X 0,Y 239.468,Z 723.326,A -85,B 0,C 180,E1 21039.643,E2 21039.643} C_VEL
LIN {X 0,Y 237.67,Z 712,A -85,B 0,C 180,E1 21046.424,E2 21046.424} C_VEL
LIN {X 0,Y 236.425,Z 703.933,A -85,B 0,C 180,E1 21054.481,E2 21054.481} C_VEL
LIN {X 0,Y 236.429,Z 702.21,A -85,B 0,C 180,E1 21059.993,E2 21059.993} C_VEL
LIN {X 0,Y 236.832,Z 702.84,A -85,B 0,C 180,E1 21063.659,E2 21063.659} C_VEL
LIN {X 0,Y 238.558,Z 711.88,A -85,B 0,C 180,E1 21072.827,E2 21072.827} C_VEL
LIN {X 0,Y 241.27,Z 724.131,A -85,B 0,C 180,E1 21079.991,E2 21079.991} C_VEL
LIN {X 0,Y 243.347,Z 739.572,A -85,B 0,C 180,E1 21086.344,E2 21086.344} C_VEL
LIN {X 0,Y 243.56,Z 751.465,A -85,B 0,C 180,E1 21090.274,E2 21090.274} C_VEL
LIN {X 0,Y 226.514,Z 780.795,A -85,B 0,C 180,E1 21094.705,E2 21094.705} C_VEL
LIN {X 0,Y 206.843,Z 808.758,A -85,B 0,C 180,E1 21101.531,E2 21101.531} C_VEL
LIN {X 0,Y 189.558,Z 830.31,A -85,B 0,C 180,E1 21110.284,E2 21110.284} C_VEL
LIN {X 0,Y 177.052,Z 845.68,A -85,B 0,C 180,E1 21120.547,E2 21120.547} C_VEL
LIN {X 0,Y 170.106,Z 855.433,A -85,B 0,C 180,E1 21131.849,E2 21131.849} C_VEL
LIN {X 0,Y 167.752,Z 860.272,A -85,B 0,C 180,E1 21143.028,E2 21143.028} C_VEL
LIN {X 0,Y 167.916,Z 861.204,A -85,B 0,C 180,E1 21150,E2 21150} C_VEL
LIN {X 0,Y 168.171,Z 859.349,A -85,B 0,C 180,E1 21160.373,E2 21160.373} C_VEL
LIN {X 0,Y 171.888,Z 852.676,A -85,B 0,C 180,E1 21172.05,E2 21172.05} C_VEL
LIN {X 0,Y 181.804,Z 839.795,A -85,B 0,C 180,E1 21184.059,E2 21184.059} C_VEL
LIN {X 0,Y 197.714,Z 820.318,A -85,B 0,C 180,E1 21194.329,E2 21194.329} C_VEL
LIN {X 0,Y 214.993,Z 797.685,A -85,B 0,C 180,E1 21201.579,E2 21201.579} C_VEL
LIN {X 0,Y 233.856,Z 769.027,A -85,B 0,C 180,E1 21207.316,E2 21207.316} C_VEL
LIN {X 0,Y 243.539,Z 751.48,A -85,B 0,C 180,E1 21209.729,E2 21209.729} C_VEL
LIN {X 0,Y 243.058,Z 736.617,A -85,B 0,C 180,E1 21214.75,E2 21214.75} C_VEL
LIN {X 0,Y 240.975,Z 722.384,A -85,B 0,C 180,E1 21220.842,E2 21220.842} C_VEL
LIN {X 0,Y 238.249,Z 710.68,A -85,B 0,C 180,E1 21228.088,E2 21228.088} C_VEL
LIN {X 0,Y 236.816,Z 702.875,A -85,B 0,C 180,E1 21236.341,E2 21236.341} C_VEL
LIN {X 0,Y 236.479,Z 702.721,A -85,B 0,C 180,E1 21243.677,E2 21243.677} C_VEL
LIN {X 0,Y 237.337,Z 710.587,A -85,B 0,C 180,E1 21252.387,E2 21252.387} C_VEL
LIN {X 0,Y 239.196,Z 721.517,A -85,B 0,C 180,E1 21259.416,E2 21259.416} C_VEL
LIN {X 0,Y 251.479,Z 746.682,A -85,B 0,C 180,E1 21274.107,E2 21274.107} C_VEL
LIN {X 0,Y 264.372,Z 760.863,A -85,B 0,C 180,E1 21282.332,E2 21282.332} C_VEL
LIN {X 0,Y 273.443,Z 770.553,A -85,B 0,C 180,E1 21288.36,E2 21288.36} C_VEL
LIN {X 0,Y 282.21,Z 779.779,A -85,B 0,C 180,E1 21294.847,E2 21294.847} C_VEL
LIN {X 0,Y 285.339,Z 782.522,A -85,B 0,C 180,E1 21297.194,E2 21297.194} C_VEL
LIN {X 0,Y 286.315,Z 787.275,A -85,B 0,C 180,E1 21299.644,E2 21299.644} C_VEL
LIN {X 0,Y 286.305,Z 794.706,A -85,B 0,C 180,E1 21303.328,E2 21303.328} C_VEL
LIN {X 0,Y 286.708,Z 795.102,A -85,B 0,C 180,E1 21303.751,E2 21303.751} C_VEL
LIN {X 0,Y 291.548,Z 800.103,A -85,B 0,C 180,E1 21309.2,E2 21309.2} C_VEL
LIN {X 0,Y 296.563,Z 804.356,A -85,B 0,C 180,E1 21315.946,E2 21315.946} C_VEL
LIN {X 0,Y 299.958,Z 805.822,A -85,B 0,C 180,E1 21321.29,E2 21321.29} C_VEL
LIN {X 0,Y 301.483,Z 807.038,A -85,B 0,C 180,E1 21327.121,E2 21327.121} C_VEL
LIN {X 0,Y 301.381,Z 807.151,A -85,B 0,C 180,E1 21332.88,E2 21332.88} C_VEL
LIN {X 0,Y 300.043,Z 805.845,A -85,B 0,C 180,E1 21338.707,E2 21338.707} C_VEL
LIN {X 0,Y 295.954,Z 804.071,A -85,B 0,C 180,E1 21344.821,E2 21344.821} C_VEL
LIN {X 0,Y 291.198,Z 799.646,A -85,B 0,C 180,E1 21351.343,E2 21351.343} C_VEL
LIN {X 0,Y 286.152,Z 794.598,A -85,B 0,C 180,E1 21356.816,E2 21356.816} C_VEL
LIN {X 0,Y 278.226,Z 786.665,A -85,B 0,C 180,E1 21363.788,E2 21363.788} C_VEL
LIN {X 0,Y 269.198,Z 777.38,A -85,B 0,C 180,E1 21370.604,E2 21370.604} C_VEL
LIN {X 0,Y 260.073,Z 767.868,A -85,B 0,C 180,E1 21376.723,E2 21376.723} C_VEL
LIN {X 0,Y 246.794,Z 753.358,A -85,B 0,C 180,E1 21385.419,E2 21385.419} C_VEL
LIN {X 0,Y 234.679,Z 726.72,A -85,B 0,C 180,E1 21401.651,E2 21401.651} C_VEL
LIN {X 0,Y 233.593,Z 717.861,A -85,B 0,C 180,E1 21407.493,E2 21407.493} C_VEL
LIN {X 0,Y 233.082,Z 709.958,A -85,B 0,C 180,E1 21416.269,E2 21416.269} C_VEL
LIN {X 0,Y 233.4,Z 710.134,A -85,B 0,C 180,E1 21423.712,E2 21423.712} C_VEL
LIN {X 0,Y 234.824,Z 719.097,A -85,B 0,C 180,E1 21432.804,E2 21432.804} C_VEL
LIN {X 0,Y 236.966,Z 731.374,A -85,B 0,C 180,E1 21439.996,E2 21439.996} C_VEL
LIN {X 0,Y 238.17,Z 746.773,A -85,B 0,C 180,E1 21446.414,E2 21446.414} C_VEL
LIN {X 0,Y 238.278,Z 753.082,A -85,B 0,C 180,E1 21448.689,E2 21448.689} C_VEL
LIN {X 0,Y 221.543,Z 781.254,A -85,B 0,C 180,E1 21453.133,E2 21453.133} C_VEL
LIN {X 0,Y 201.582,Z 808.52,A -85,B 0,C 180,E1 21459.813,E2 21459.813} C_VEL
LIN {X 0,Y 183.409,Z 830.071,A -85,B 0,C 180,E1 21468.669,E2 21468.669} C_VEL
LIN {X 0,Y 170.043,Z 845.44,A -85,B 0,C 180,E1 21479.205,E2 21479.205} C_VEL
LIN {X 0,Y 162.482,Z 855.195,A -85,B 0,C 180,E1 21490.965,E2 21490.965} C_VEL
LIN {X 0,Y 160.323,Z 859.113,A -85,B 0,C 180,E1 21499.113,E2 21499.113} C_VEL
LIN {X 0,Y 160.028,Z 860.971,A -85,B 0,C 180,E1 21510,E2 21510} C_VEL
LIN {X 0,Y 160.324,Z 859.113,A -85,B 0,C 180,E1 21520.887,E2 21520.887} C_VEL
LIN {X 0,Y 164.338,Z 852.588,A -85,B 0,C 180,E1 21532.912,E2 21532.912} C_VEL
LIN {X 0,Y 175.342,Z 839.299,A -85,B 0,C 180,E1 21545.731,E2 21545.731} C_VEL
LIN {X 0,Y 191.997,Z 820.078,A -85,B 0,C 180,E1 21556.02,E2 21556.02} C_VEL
LIN {X 0,Y 210.062,Z 797.446,A -85,B 0,C 180,E1 21563.307,E2 21563.307} C_VEL
LIN {X 0,Y 229.616,Z 768.79,A -85,B 0,C 180,E1 21569.004,E2 21569.004} C_VEL
LIN {X 0,Y 238.269,Z 753.063,A -85,B 0,C 180,E1 21571.321,E2 21571.321} C_VEL
LIN {X 0,Y 237.439,Z 735.3,A -85,B 0,C 180,E1 21578.145,E2 21578.145} C_VEL
LIN {X 0,Y 235.399,Z 722.103,A -85,B 0,C 180,E1 21585.099,E2 21585.099} C_VEL
LIN {X 0,Y 233.984,Z 715.032,A -85,B 0,C 180,E1 21590.698,E2 21590.698} C_VEL
LIN {X 0,Y 233.39,Z 710.155,A -85,B 0,C 180,E1 21596.287,E2 21596.287} C_VEL
LIN {X 0,Y 233.073,Z 709.978,A -85,B 0,C 180,E1 21603.731,E2 21603.731} C_VEL
LIN {X 0,Y 233.58,Z 717.87,A -85,B 0,C 180,E1 21612.497,E2 21612.497} C_VEL
LIN {X 0,Y 235.271,Z 730.833,A -85,B 0,C 180,E1 21620.735,E2 21620.735} C_VEL
LIN {X 0,Y 252.04,Z 759.009,A -85,B 0,C 180,E1 21638.135,E2 21638.135} C_VEL
LIN {X 0,Y 263.71,Z 771.372,A -85,B 0,C 180,E1 21645.554,E2 21645.554} C_VEL
LIN {X 0,Y 273.334,Z 781.782,A -85,B 0,C 180,E1 21652.46,E2 21652.46} C_VEL
LIN {X 0,Y 281.823,Z 790.377,A -85,B 0,C 180,E1 21659.276,E2 21659.276} C_VEL
LIN {X 0,Y 286.708,Z 795.102,A -85,B 0,C 180,E1 21663.751,E2 21663.751} C_VEL
LIN {X 0,Y 287.281,Z 799.037,A -85,B 0,C 180,E1 21666.249,E2 21666.249} C_VEL
LIN {X 0,Y 286.073,Z 805.705,A -85,B 0,C 180,E1 21670.015,E2 21670.015} C_VEL
LIN {X 0,Y 286.304,Z 806.079,A -85,B 0,C 180,E1 21670.451,E2 21670.451} C_VEL
LIN {X 0,Y 289.64,Z 808.883,A -85,B 0,C 180,E1 21674.849,E2 21674.849} C_VEL
LIN {X 0,Y 293.739,Z 810.834,A -85,B 0,C 180,E1 21681.104,E2 21681.104} C_VEL
LIN {X 0,Y 295.397,Z 812.062,A -85,B 0,C 180,E1 21687.062,E2 21687.062} C_VEL
LIN {X 0,Y 295.294,Z 812.174,A -85,B 0,C 180,E1 21692.939,E2 21692.939} C_VEL
LIN {X 0,Y 293.818,Z 810.866,A -85,B 0,C 180,E1 21698.893,E2 21698.893} C_VEL
LIN {X 0,Y 289.528,Z 808.882,A -85,B 0,C 180,E1 21705.157,E2 21705.157} C_VEL
LIN {X 0,Y 284.696,Z 804.137,A -85,B 0,C 180,E1 21711.856,E2 21711.856} C_VEL
LIN {X 0,Y 279.966,Z 799.539,A -85,B 0,C 180,E1 21716.869,E2 21716.869} C_VEL
LIN {X 0,Y 272.107,Z 791.652,A -85,B 0,C 180,E1 21723.808,E2 21723.808} C_VEL
LIN {X 0,Y 263.165,Z 782.459,A -85,B 0,C 180,E1 21730.596,E2 21730.596} C_VEL
LIN {X 0,Y 254.528,Z 773.434,A -85,B 0,C 180,E1 21736.427,E2 21736.427} C_VEL
LIN {X 0,Y 240.021,Z 757.638,A -85,B 0,C 180,E1 21746.391,E2 21746.391} C_VEL
LIN {X 0,Y 230.042,Z 731.789,A -85,B 0,C 180,E1 21762.766,E2 21762.766} C_VEL
LIN {X 0,Y 229.506,Z 723.654,A -85,B 0,C 180,E1 21768.579,E2 21768.579} C_VEL
LIN {X 0,Y 229.485,Z 717.16,A -85,B 0,C 180,E1 21776.21,E2 21776.21} C_VEL
LIN {X 0,Y 229.597,Z 716.466,A -85,B 0,C 180,E1 21779.993,E2 21779.993} C_VEL
LIN {X 0,Y 229.756,Z 718.614,A -85,B 0,C 180,E1 21785.338,E2 21785.338} C_VEL
LIN {X 0,Y 230.873,Z 726.537,A -85,B 0,C 180,E1 21793.027,E2 21793.027} C_VEL
LIN {X 0,Y 232.295,Z 738.394,A -85,B 0,C 180,E1 21800.002,E2 21800.002} C_VEL
LIN {X 0,Y 232.763,Z 755.349,A -85,B 0,C 180,E1 21807.077,E2 21807.077} C_VEL
LIN {X 0,Y 231.202,Z 759.313,A -85,B 0,C 180,E1 21807.962,E2 21807.962} C_VEL
LIN {X 0,Y 211.806,Z 788.644,A -85,B 0,C 180,E1 21812.868,E2 21812.868} C_VEL
LIN {X 0,Y 192.029,Z 813.457,A -85,B 0,C 180,E1 21819.759,E2 21819.759} C_VEL
LIN {X 0,Y 175.552,Z 831.892,A -85,B 0,C 180,E1 21828.056,E2 21828.056} C_VEL
LIN {X 0,Y 161.921,Z 846.476,A -85,B 0,C 180,E1 21839.051,E2 21839.051} C_VEL
LIN {X 0,Y 153.83,Z 856.556,A -85,B 0,C 180,E1 21852.826,E2 21852.826} C_VEL
LIN {X 0,Y 151.906,Z 860.359,A -85,B 0,C 180,E1 21865.193,E2 21865.193} C_VEL
LIN {X 0,Y 152.118,Z 860.738,A -85,B 0,C 180,E1 21870,E2 21870} C_VEL
LIN {X 0,Y 152.504,Z 858.877,A -85,B 0,C 180,E1 21881.453,E2 21881.453} C_VEL
LIN {X 0,Y 156.908,Z 852.349,A -85,B 0,C 180,E1 21894.064,E2 21894.064} C_VEL
LIN {X 0,Y 167.727,Z 840.205,A -85,B 0,C 180,E1 21906.442,E2 21906.442} C_VEL
LIN {X 0,Y 184.108,Z 822.473,A -85,B 0,C 180,E1 21916.669,E2 21916.669} C_VEL
LIN {X 0,Y 202.946,Z 800.336,A -85,B 0,C 180,E1 21924.319,E2 21924.319} C_VEL
LIN {X 0,Y 222.504,Z 773.248,A -85,B 0,C 180,E1 21929.977,E2 21929.977} C_VEL
LIN {X 0,Y 232.731,Z 756.117,A -85,B 0,C 180,E1 21932.647,E2 21932.647} C_VEL
LIN {X 0,Y 232.435,Z 739.331,A -85,B 0,C 180,E1 21939.513,E2 21939.513} C_VEL
LIN {X 0,Y 231.146,Z 728.033,A -85,B 0,C 180,E1 21945.902,E2 21945.902} C_VEL
LIN {X 0,Y 229.84,Z 720.554,A -85,B 0,C 180,E1 21952.437,E2 21952.437} C_VEL
LIN {X 0,Y 229.832,Z 717.38,A -85,B 0,C 180,E1 21956.23,E2 21956.23} C_VEL
LIN {X 0,Y 229.601,Z 716.459,A -85,B 0,C 180,E1 21960.007,E2 21960.007} C_VEL
LIN {X 0,Y 229.287,Z 718.511,A -85,B 0,C 180,E1 21965.773,E2 21965.773} C_VEL
LIN {X 0,Y 229.806,Z 726.884,A -85,B 0,C 180,E1 21974.011,E2 21974.011} C_VEL
LIN {X 0,Y 238.924,Z 756.047,A -85,B 0,C 180,E1 21992.598,E2 21992.598} C_VEL
LIN {X 0,Y 252.936,Z 771.732,A -85,B 0,C 180,E1 22002.548,E2 22002.548} C_VEL
LIN {X 0,Y 262.08,Z 781.471,A -85,B 0,C 180,E1 22008.685,E2 22008.685} C_VEL
LIN {X 0,Y 270.811,Z 790.611,A -85,B 0,C 180,E1 22015.246,E2 22015.246} C_VEL
LIN {X 0,Y 278.364,Z 798.258,A -85,B 0,C 180,E1 22021.752,E2 22021.752} C_VEL
LIN {X 0,Y 283.462,Z 802.64,A -85,B 0,C 180,E1 22026.55,E2 22026.55} C_VEL
LIN {X 0,Y 286.304,Z 806.079,A -85,B 0,C 180,E1 22030.451,E2 22030.451} C_VEL
LIN {X 0,Y 285.486,Z 810.811,A -85,B 0,C 180,E1 22033.839,E2 22033.839} C_VEL
LIN {X 0,Y 284.874,Z 814.547,A -85,B 0,C 180,E1 22037.282,E2 22037.282} C_VEL
LIN {X 0,Y 287.295,Z 815.577,A -85,B 0,C 180,E1 22040.903,E2 22040.903} C_VEL
LIN {X 0,Y 289.04,Z 816.751,A -85,B 0,C 180,E1 22046.997,E2 22046.997} C_VEL
LIN {X 0,Y 288.928,Z 816.862,A -85,B 0,C 180,E1 22053.004,E2 22053.004} C_VEL
LIN {X 0,Y 287.384,Z 815.604,A -85,B 0,C 180,E1 22059.094,E2 22059.094} C_VEL
LIN {X 0,Y 282.864,Z 813.367,A -85,B 0,C 180,E1 22065.523,E2 22065.523} C_VEL
LIN {X 0,Y 277.898,Z 808.346,A -85,B 0,C 180,E1 22072.419,E2 22072.419} C_VEL
LIN {X 0,Y 270.964,Z 801.823,A -85,B 0,C 180,E1 22079.299,E2 22079.299} C_VEL
LIN {X 0,Y 264.302,Z 795.032,A -85,B 0,C 180,E1 22084.949,E2 22084.949} C_VEL
LIN {X 0,Y 255.739,Z 786.116,A -85,B 0,C 180,E1 22091.391,E2 22091.391} C_VEL
LIN {X 0,Y 245.673,Z 775.38,A -85,B 0,C 180,E1 22098.178,E2 22098.178} C_VEL
LIN {X 0,Y 227.153,Z 749.961,A -85,B 0,C 180,E1 22115.583,E2 22115.583} C_VEL
LIN {X 0,Y 225.374,Z 731.987,A -85,B 0,C 180,E1 22127.382,E2 22127.382} C_VEL
LIN {X 0,Y 225.646,Z 724.224,A -85,B 0,C 180,E1 22136.146,E2 22136.146} C_VEL
LIN {X 0,Y 225.822,Z 723.396,A -85,B 0,C 180,E1 22139.993,E2 22139.993} C_VEL
LIN {X 0,Y 225.896,Z 725.732,A -85,B 0,C 180,E1 22145.43,E2 22145.43} C_VEL
LIN {X 0,Y 226.71,Z 734.15,A -85,B 0,C 180,E1 22153.51,E2 22153.51} C_VEL
LIN {X 0,Y 227.474,Z 746.216,A -85,B 0,C 180,E1 22160.445,E2 22160.445} C_VEL
LIN {X 0,Y 226.834,Z 760.242,A -85,B 0,C 180,E1 22166.338,E2 22166.338} C_VEL
LIN {X 0,Y 207.56,Z 788.407,A -85,B 0,C 180,E1 22171.006,E2 22171.006} C_VEL
LIN {X 0,Y 186.969,Z 813.218,A -85,B 0,C 180,E1 22177.857,E2 22177.857} C_VEL
LIN {X 0,Y 169.608,Z 831.652,A -85,B 0,C 180,E1 22186.225,E2 22186.225} C_VEL
LIN {X 0,Y 155.033,Z 846.237,A -85,B 0,C 180,E1 22197.512,E2 22197.512} C_VEL
LIN {X 0,Y 146.172,Z 856.318,A -85,B 0,C 180,E1 22211.896,E2 22211.896} C_VEL
LIN {X 0,Y 144.052,Z 860.031,A -85,B 0,C 180,E1 22223.967,E2 22223.967} C_VEL
LIN {X 0,Y 144.209,Z 860.504,A -85,B 0,C 180,E1 22230,E2 22230} C_VEL
LIN {X 0,Y 144.677,Z 858.641,A -85,B 0,C 180,E1 22242.081,E2 22242.081} C_VEL
LIN {X 0,Y 150.559,Z 850.975,A -85,B 0,C 180,E1 22256.906,E2 22256.906} C_VEL
LIN {X 0,Y 162.367,Z 838.909,A -85,B 0,C 180,E1 22269.008,E2 22269.008} C_VEL
LIN {X 0,Y 181.131,Z 819.6,A -85,B 0,C 180,E1 22279.707,E2 22279.707} C_VEL
LIN {X 0,Y 200.831,Z 796.968,A -85,B 0,C 180,E1 22287.004,E2 22287.004} C_VEL
LIN {X 0,Y 221.786,Z 768.316,A -85,B 0,C 180,E1 22292.556,E2 22292.556} C_VEL
LIN {X 0,Y 227.132,Z 759.053,A -85,B 0,C 180,E1 22294.036,E2 22294.036} C_VEL
LIN {X 0,Y 227.488,Z 744.138,A -85,B 0,C 180,E1 22300.571,E2 22300.571} C_VEL
LIN {X 0,Y 226.572,Z 732.859,A -85,B 0,C 180,E1 22307.464,E2 22307.464} C_VEL
LIN {X 0,Y 225.992,Z 724.445,A -85,B 0,C 180,E1 22316.166,E2 22316.166} C_VEL
LIN {X 0,Y 225.824,Z 723.392,A -85,B 0,C 180,E1 22320.007,E2 22320.007} C_VEL
LIN {X 0,Y 225.413,Z 725.623,A -85,B 0,C 180,E1 22325.872,E2 22325.872} C_VEL
LIN {X 0,Y 225.393,Z 733.264,A -85,B 0,C 180,E1 22333.605,E2 22333.605} C_VEL
LIN {X 0,Y 232.278,Z 760.101,A -85,B 0,C 180,E1 22351.437,E2 22351.437} C_VEL
LIN {X 0,Y 246.767,Z 776.664,A -85,B 0,C 180,E1 22362.586,E2 22362.586} C_VEL
LIN {X 0,Y 255.659,Z 786.129,A -85,B 0,C 180,E1 22368.605,E2 22368.605} C_VEL
LIN {X 0,Y 265.332,Z 796.071,A -85,B 0,C 180,E1 22375.874,E2 22375.874} C_VEL
LIN {X 0,Y 272.919,Z 803.753,A -85,B 0,C 180,E1 22382.584,E2 22382.584} C_VEL
LIN {X 0,Y 278.035,Z 808.48,A -85,B 0,C 180,E1 22387.79,E2 22387.79} C_VEL
LIN {X 0,Y 282.96,Z 813.391,A -85,B 0,C 180,E1 22394.482,E2 22394.482} C_VEL
LIN {X 0,Y 284.874,Z 814.547,A -85,B 0,C 180,E1 22397.282,E2 22397.282} C_VEL
LIN {X 0,Y 284.659,Z 816.857,A -85,B 0,C 180,E1 22399.873,E2 22399.873} C_VEL
LIN {X 0,Y 281.86,Z 820.775,A -85,B 0,C 180,E1 22404.256,E2 22404.256} C_VEL
LIN {X 0,Y 282.574,Z 821.459,A -85,B 0,C 180,E1 22410,E2 22410} C_VEL
LIN {X 0,Y 281.929,Z 820.695,A -85,B 0,C 180,E1 22416.166,E2 22416.166} C_VEL
LIN {X 0,Y 278.809,Z 819.271,A -85,B 0,C 180,E1 22422.168,E2 22422.168} C_VEL
LIN {X 0,Y 273.354,Z 815.132,A -85,B 0,C 180,E1 22429.668,E2 22429.668} C_VEL
LIN {X 0,Y 268.497,Z 810.001,A -85,B 0,C 180,E1 22435.537,E2 22435.537} C_VEL
LIN {X 0,Y 261.443,Z 802.969,A -85,B 0,C 180,E1 22442.069,E2 22442.069} C_VEL
LIN {X 0,Y 252.823,Z 794.141,A -85,B 0,C 180,E1 22448.868,E2 22448.868} C_VEL
LIN {X 0,Y 243.227,Z 784.209,A -85,B 0,C 180,E1 22455.542,E2 22455.542} C_VEL
LIN {X 0,Y 228.315,Z 768.141,A -85,B 0,C 180,E1 22466.8,E2 22466.8} C_VEL
LIN {X 0,Y 220.718,Z 743.44,A -85,B 0,C 180,E1 22484.068,E2 22484.068} C_VEL
LIN {X 0,Y 221.009,Z 735.839,A -85,B 0,C 180,E1 22490.132,E2 22490.132} C_VEL
LIN {X 0,Y 221.572,Z 731.175,A -85,B 0,C 180,E1 22496.075,E2 22496.075} C_VEL
LIN {X 0,Y 221.898,Z 730.254,A -85,B 0,C 180,E1 22499.993,E2 22499.993} C_VEL
LIN {X 0,Y 221.768,Z 732.991,A -85,B 0,C 180,E1 22505.87,E2 22505.87} C_VEL
LIN {X 0,Y 222.216,Z 740.169,A -85,B 0,C 180,E1 22512.877,E2 22512.877} C_VEL
LIN {X 0,Y 222.342,Z 751.879,A -85,B 0,C 180,E1 22519.898,E2 22519.898} C_VEL
LIN {X 0,Y 221.534,Z 762.896,A -85,B 0,C 180,E1 22524.866,E2 22524.866} C_VEL
LIN {X 0,Y 201.53,Z 790.678,A -85,B 0,C 180,E1 22529.605,E2 22529.605} C_VEL
LIN {X 0,Y 179.299,Z 816.002,A -85,B 0,C 180,E1 22536.931,E2 22536.931} C_VEL
LIN {X 0,Y 159.892,Z 835.11,A -85,B 0,C 180,E1 22546.645,E2 22546.645} C_VEL
LIN {X 0,Y 145.661,Z 848.548,A -85,B 0,C 180,E1 22558.687,E2 22558.687} C_VEL
LIN {X 0,Y 137.586,Z 857.269,A -85,B 0,C 180,E1 22574.031,E2 22574.031} C_VEL
LIN {X 0,Y 136.155,Z 859.797,A -85,B 0,C 180,E1 22583.615,E2 22583.615} C_VEL
LIN {X 0,Y 136.238,Z 860.242,A -85,B 0,C 180,E1 22590.554,E2 22590.554} C_VEL
LIN {X 0,Y 136.888,Z 858.405,A -85,B 0,C 180,E1 22602.78,E2 22602.78} C_VEL
LIN {X 0,Y 143.415,Z 850.736,A -85,B 0,C 180,E1 22618.364,E2 22618.364} C_VEL
LIN {X 0,Y 156.158,Z 838.669,A -85,B 0,C 180,E1 22630.879,E2 22630.879} C_VEL
LIN {X 0,Y 175.904,Z 819.458,A -85,B 0,C 180,E1 22641.676,E2 22641.676} C_VEL
LIN {X 0,Y 196.463,Z 796.854,A -85,B 0,C 180,E1 22648.943,E2 22648.943} C_VEL
LIN {X 0,Y 218.222,Z 768.08,A -85,B 0,C 180,E1 22654.417,E2 22654.417} C_VEL
LIN {X 0,Y 221.507,Z 762.902,A -85,B 0,C 180,E1 22655.146,E2 22655.146} C_VEL
LIN {X 0,Y 222.411,Z 748.532,A -85,B 0,C 180,E1 22661.814,E2 22661.814} C_VEL
LIN {X 0,Y 222.065,Z 737.517,A -85,B 0,C 180,E1 22669.201,E2 22669.201} C_VEL
LIN {X 0,Y 221.958,Z 731.425,A -85,B 0,C 180,E1 22676.096,E2 22676.096} C_VEL
LIN {X 0,Y 221.901,Z 730.25,A -85,B 0,C 180,E1 22680.007,E2 22680.007} C_VEL
LIN {X 0,Y 221.265,Z 732.496,A -85,B 0,C 180,E1 22685.898,E2 22685.898} C_VEL
LIN {X 0,Y 220.944,Z 739.341,A -85,B 0,C 180,E1 22693.006,E2 22693.006} C_VEL
LIN {X 0,Y 227.386,Z 766.706,A -85,B 0,C 180,E1 22712.194,E2 22712.194} C_VEL
LIN {X 0,Y 240.427,Z 781.323,A -85,B 0,C 180,E1 22722.612,E2 22722.612} C_VEL
LIN {X 0,Y 249.854,Z 791.368,A -85,B 0,C 180,E1 22729.083,E2 22729.083} C_VEL
LIN {X 0,Y 259.666,Z 801.32,A -85,B 0,C 180,E1 22736.495,E2 22736.495} C_VEL
LIN {X 0,Y 266.846,Z 808.606,A -85,B 0,C 180,E1 22743.005,E2 22743.005} C_VEL
LIN {X 0,Y 272.374,Z 813.969,A -85,B 0,C 180,E1 22748.92,E2 22748.92} C_VEL
LIN {X 0,Y 276.078,Z 817.582,A -85,B 0,C 180,E1 22754.085,E2 22754.085} C_VEL
LIN {X 0,Y 280.561,Z 819.979,A -85,B 0,C 180,E1 22760.683,E2 22760.683} C_VEL
LIN {X 0,Y 281.86,Z 820.775,A -85,B 0,C 180,E1 22764.256,E2 22764.256} C_VEL
LIN {X 0,Y 280.105,Z 822.792,A -85,B 0,C 180,E1 22766.877,E2 22766.877} C_VEL
LIN {X 0,Y 275.713,Z 825.565,A -85,B 0,C 180,E1 22771.293,E2 22771.293} C_VEL
LIN {X 0,Y 274.724,Z 824.7,A -85,B 0,C 180,E1 22777.219,E2 22777.219} C_VEL
LIN {X 0,Y 271.443,Z 823.132,A -85,B 0,C 180,E1 22782.892,E2 22782.892} C_VEL
LIN {X 0,Y 266.398,Z 818.993,A -85,B 0,C 180,E1 22789.938,E2 22789.938} C_VEL
LIN {X 0,Y 260.864,Z 813.381,A -85,B 0,C 180,E1 22796.341,E2 22796.341} C_VEL
LIN {X 0,Y 253.308,Z 805.798,A -85,B 0,C 180,E1 22803.189,E2 22803.189} C_VEL
LIN {X 0,Y 245.095,Z 797.36,A -85,B 0,C 180,E1 22809.6,E2 22809.6} C_VEL
LIN {X 0,Y 234.134,Z 786.068,A -85,B 0,C 180,E1 22817.228,E2 22817.228} C_VEL
LIN {X 0,Y 218.359,Z 766.69,A -85,B 0,C 180,E1 22832.073,E2 22832.073} C_VEL
LIN {X 0,Y 216.366,Z 744.319,A -85,B 0,C 180,E1 22848.428,E2 22848.428} C_VEL
LIN {X 0,Y 217.318,Z 738.025,A -85,B 0,C 180,E1 22855.998,E2 22855.998} C_VEL
LIN {X 0,Y 217.711,Z 736.982,A -85,B 0,C 180,E1 22859.993,E2 22859.993} C_VEL
LIN {X 0,Y 217.524,Z 739.475,A -85,B 0,C 180,E1 22865.47,E2 22865.47} C_VEL
LIN {X 0,Y 217.511,Z 746.979,A -85,B 0,C 180,E1 22872.964,E2 22872.964} C_VEL
LIN {X 0,Y 217.005,Z 758.353,A -85,B 0,C 180,E1 22879.816,E2 22879.816} C_VEL
LIN {X 0,Y 215.648,Z 766.729,A -85,B 0,C 180,E1 22883.493,E2 22883.493} C_VEL
LIN {X 0,Y 193.292,Z 795.569,A -85,B 0,C 180,E1 22888.745,E2 22888.745} C_VEL
LIN {X 0,Y 171.969,Z 818.297,A -85,B 0,C 180,E1 22895.798,E2 22895.798} C_VEL
LIN {X 0,Y 152.086,Z 836.654,A -85,B 0,C 180,E1 22905.824,E2 22905.824} C_VEL
LIN {X 0,Y 137.542,Z 849.462,A -85,B 0,C 180,E1 22918.475,E2 22918.475} C_VEL
LIN {X 0,Y 129.89,Z 857.031,A -85,B 0,C 180,E1 22933.058,E2 22933.058} C_VEL
LIN {X 0,Y 128.253,Z 859.562,A -85,B 0,C 180,E1 22943.22,E2 22943.22} C_VEL
LIN {X 0,Y 128.42,Z 860.037,A -85,B 0,C 180,E1 22950,E2 22950} C_VEL
LIN {X 0,Y 129.098,Z 858.169,A -85,B 0,C 180,E1 22963.566,E2 22963.566} C_VEL
LIN {X 0,Y 136.348,Z 850.497,A -85,B 0,C 180,E1 22979.98,E2 22979.98} C_VEL
LIN {X 0,Y 150.117,Z 838.43,A -85,B 0,C 180,E1 22992.906,E2 22992.906} C_VEL
LIN {X 0,Y 169.862,Z 820.297,A -85,B 0,C 180,E1 23003.342,E2 23003.342} C_VEL
LIN {X 0,Y 191.112,Z 798.181,A -85,B 0,C 180,E1 23010.629,E2 23010.629} C_VEL
LIN {X 0,Y 214.11,Z 768.906,A -85,B 0,C 180,E1 23016.186,E2 23016.186} C_VEL
LIN {X 0,Y 216.191,Z 765.545,A -85,B 0,C 180,E1 23016.793,E2 23016.793} C_VEL
LIN {X 0,Y 217.405,Z 753.341,A -85,B 0,C 180,E1 23022.898,E2 23022.898} C_VEL
LIN {X 0,Y 217.552,Z 743.436,A -85,B 0,C 180,E1 23029.988,E2 23029.988} C_VEL
LIN {X 0,Y 217.687,Z 738.302,A -85,B 0,C 180,E1 23036.019,E2 23036.019} C_VEL
LIN {X 0,Y 217.713,Z 736.979,A -85,B 0,C 180,E1 23040.007,E2 23040.007} C_VEL
LIN {X 0,Y 217.01,Z 739.251,A -85,B 0,C 180,E1 23045.812,E2 23045.812} C_VEL
LIN {X 0,Y 216.149,Z 746.426,A -85,B 0,C 180,E1 23053.3,E2 23053.3} C_VEL
LIN {X 0,Y 221.462,Z 771.851,A -85,B 0,C 180,E1 23072.002,E2 23072.002} C_VEL
LIN {X 0,Y 234.14,Z 786.062,A -85,B 0,C 180,E1 23082.771,E2 23082.771} C_VEL
LIN {X 0,Y 244.998,Z 797.412,A -85,B 0,C 180,E1 23090.389,E2 23090.389} C_VEL
LIN {X 0,Y 254.251,Z 806.739,A -85,B 0,C 180,E1 23097.592,E2 23097.592} C_VEL
LIN {X 0,Y 261.693,Z 814.104,A -85,B 0,C 180,E1 23104.481,E2 23104.481} C_VEL
LIN {X 0,Y 266.388,Z 818.977,A -85,B 0,C 180,E1 23110.061,E2 23110.061} C_VEL
LIN {X 0,Y 271.47,Z 823.148,A -85,B 0,C 180,E1 23117.109,E2 23117.109} C_VEL
LIN {X 0,Y 274.692,Z 824.758,A -85,B 0,C 180,E1 23122.833,E2 23122.833} C_VEL
LIN {X 0,Y 275.795,Z 825.375,A -85,B 0,C 180,E1 23126.853,E2 23126.853} C_VEL
LIN {X 0,Y 275.713,Z 825.565,A -85,B 0,C 180,E1 23131.293,E2 23131.293} C_VEL
LIN {X 0,Y 273.201,Z 826.752,A -85,B 0,C 180,E1 23133.967,E2 23133.967} C_VEL
LIN {X 0,Y 267.15,Z 828.261,A -85,B 0,C 180,E1 23138.475,E2 23138.475} C_VEL
LIN {X 0,Y 264.205,Z 826.793,A -85,B 0,C 180,E1 23143.251,E2 23143.251} C_VEL
LIN {X 0,Y 258.933,Z 822.242,A -85,B 0,C 180,E1 23150.669,E2 23150.669} C_VEL
LIN {X 0,Y 252.85,Z 816.295,A -85,B 0,C 180,E1 23157.303,E2 23157.303} C_VEL
LIN {X 0,Y 245.722,Z 809.103,A -85,B 0,C 180,E1 23163.68,E2 23163.68} C_VEL
LIN {X 0,Y 236.438,Z 799.586,A -85,B 0,C 180,E1 23170.807,E2 23170.807} C_VEL
LIN {X 0,Y 223.969,Z 786.697,A -85,B 0,C 180,E1 23180.036,E2 23180.036} C_VEL
LIN {X 0,Y 210.269,Z 760.691,A -85,B 0,C 180,E1 23201.138,E2 23201.138} C_VEL
LIN {X 0,Y 211.744,Z 749.796,A -85,B 0,C 180,E1 23209.487,E2 23209.487} C_VEL
LIN {X 0,Y 212.795,Z 744.723,A -85,B 0,C 180,E1 23215.913,E2 23215.913} C_VEL
LIN {X 0,Y 213.348,Z 743.608,A -85,B 0,C 180,E1 23219.993,E2 23219.993} C_VEL
LIN {X 0,Y 212.965,Z 746.155,A -85,B 0,C 180,E1 23225.548,E2 23225.548} C_VEL
LIN {X 0,Y 212.664,Z 754.022,A -85,B 0,C 180,E1 23233.265,E2 23233.265} C_VEL
LIN {X 0,Y 211.367,Z 765.52,A -85,B 0,C 180,E1 23240.152,E2 23240.152} C_VEL
LIN {X 0,Y 210.865,Z 768.419,A -85,B 0,C 180,E1 23241.582,E2 23241.582} C_VEL
LIN {X 0,Y 189.257,Z 795.669,A -85,B 0,C 180,E1 23246.689,E2 23246.689} C_VEL
LIN {X 0,Y 166.871,Z 818.505,A -85,B 0,C 180,E1 23253.74,E2 23253.74} C_VEL
LIN {X 0,Y 144.329,Z 838.192,A -85,B 0,C 180,E1 23264.92,E2 23264.92} C_VEL
LIN {X 0,Y 128.175,Z 851.293,A -85,B 0,C 180,E1 23279.866,E2 23279.866} C_VEL
LIN {X 0,Y 121.33,Z 857.932,A -85,B 0,C 180,E1 23295.548,E2 23295.548} C_VEL
LIN {X 0,Y 120.508,Z 859.804,A -85,B 0,C 180,E1 23310,E2 23310} C_VEL
LIN {X 0,Y 121.331,Z 857.932,A -85,B 0,C 180,E1 23324.452,E2 23324.452} C_VEL
LIN {X 0,Y 129.415,Z 850.259,A -85,B 0,C 180,E1 23341.767,E2 23341.767} C_VEL
LIN {X 0,Y 144.296,Z 838.191,A -85,B 0,C 180,E1 23355.093,E2 23355.093} C_VEL
LIN {X 0,Y 166.863,Z 818.503,A -85,B 0,C 180,E1 23366.265,E2 23366.265} C_VEL
LIN {X 0,Y 189.298,Z 795.631,A -85,B 0,C 180,E1 23373.316,E2 23373.316} C_VEL
LIN {X 0,Y 210.716,Z 769.019,A -85,B 0,C 180,E1 23378.142,E2 23378.142} C_VEL
LIN {X 0,Y 212.396,Z 757.204,A -85,B 0,C 180,E1 23384.504,E2 23384.504} C_VEL
LIN {X 0,Y 212.806,Z 750.266,A -85,B 0,C 180,E1 23389.762,E2 23389.762} C_VEL
LIN {X 0,Y 213.185,Z 745.033,A -85,B 0,C 180,E1 23395.935,E2 23395.935} C_VEL
LIN {X 0,Y 213.36,Z 743.59,A -85,B 0,C 180,E1 23400.007,E2 23400.007} C_VEL
LIN {X 0,Y 212.355,Z 746.091,A -85,B 0,C 180,E1 23406.145,E2 23406.145} C_VEL
LIN {X 0,Y 211.193,Z 753.247,A -85,B 0,C 180,E1 23413.481,E2 23413.481} C_VEL
LIN {X 0,Y 215.452,Z 776.959,A -85,B 0,C 180,E1 23431.877,E2 23431.877} C_VEL
LIN {X 0,Y 229.136,Z 792.003,A -85,B 0,C 180,E1 23443.937,E2 23443.937} C_VEL
LIN {X 0,Y 240.024,Z 803.318,A -85,B 0,C 180,E1 23451.844,E2 23451.844} C_VEL
LIN {X 0,Y 249.127,Z 812.488,A -85,B 0,C 180,E1 23459.198,E2 23459.198} C_VEL
LIN {X 0,Y 255.782,Z 818.952,A -85,B 0,C 180,E1 23465.521,E2 23465.521} C_VEL
LIN {X 0,Y 260.39,Z 823.769,A -85,B 0,C 180,E1 23471.349,E2 23471.349} C_VEL
LIN {X 0,Y 264.32,Z 826.867,A -85,B 0,C 180,E1 23476.866,E2 23476.866} C_VEL
LIN {X 0,Y 268.087,Z 828.749,A -85,B 0,C 180,E1 23483.514,E2 23483.514} C_VEL
LIN {X 0,Y 269.014,Z 829.511,A -85,B 0,C 180,E1 23490,E2 23490} C_VEL
LIN {X 0,Y 268.22,Z 828.748,A -85,B 0,C 180,E1 23496.482,E2 23496.482} C_VEL
LIN {X 0,Y 267.15,Z 828.261,A -85,B 0,C 180,E1 23498.475,E2 23498.475} C_VEL
LIN {X 0,Y 263.334,Z 828.799,A -85,B 0,C 180,E1 23501.17,E2 23501.17} C_VEL
LIN {X 0,Y 255.295,Z 829.32,A -85,B 0,C 180,E1 23505.591,E2 23505.591} C_VEL
LIN {X 0,Y 255.206,Z 829.036,A -85,B 0,C 180,E1 23505.713,E2 23505.713} C_VEL
LIN {X 0,Y 250.245,Z 824.034,A -85,B 0,C 180,E1 23512.669,E2 23512.669} C_VEL
LIN {X 0,Y 243.057,Z 817.043,A -85,B 0,C 180,E1 23519.89,E2 23519.89} C_VEL
LIN {X 0,Y 234.656,Z 808.579,A -85,B 0,C 180,E1 23526.883,E2 23526.883} C_VEL
LIN {X 0,Y 222.768,Z 796.583,A -85,B 0,C 180,E1 23535.697,E2 23535.697} C_VEL
LIN {X 0,Y 208.428,Z 780.614,A -85,B 0,C 180,E1 23549.429,E2 23549.429} C_VEL
LIN {X 0,Y 206.723,Z 756.275,A -85,B 0,C 180,E1 23569.442,E2 23569.442} C_VEL
LIN {X 0,Y 208.109,Z 751.353,A -85,B 0,C 180,E1 23575.82,E2 23575.82} C_VEL
LIN {X 0,Y 208.781,Z 750.076,A -85,B 0,C 180,E1 23579.992,E2 23579.992} C_VEL
LIN {X 0,Y 208.3,Z 752.791,A -85,B 0,C 180,E1 23585.672,E2 23585.672} C_VEL
LIN {X 0,Y 207.544,Z 759.573,A -85,B 0,C 180,E1 23592.633,E2 23592.633} C_VEL
LIN {X 0,Y 205.67,Z 770.803,A -85,B 0,C 180,E1 23599.626,E2 23599.626} C_VEL
LIN {X 0,Y 205.334,Z 772.137,A -85,B 0,C 180,E1 23600.298,E2 23600.298} C_VEL
LIN {X 0,Y 182.232,Z 799.299,A -85,B 0,C 180,E1 23605.373,E2 23605.373} C_VEL
LIN {X 0,Y 156.717,Z 823.347,A -85,B 0,C 180,E1 23613.564,E2 23613.564} C_VEL
LIN {X 0,Y 136.599,Z 839.498,A -85,B 0,C 180,E1 23623.908,E2 23623.908} C_VEL
LIN {X 0,Y 120.029,Z 852.089,A -85,B 0,C 180,E1 23639.698,E2 23639.698} C_VEL
LIN {X 0,Y 113.597,Z 857.696,A -85,B 0,C 180,E1 23654.54,E2 23654.54} C_VEL
LIN {X 0,Y 112.591,Z 859.57,A -85,B 0,C 180,E1 23670,E2 23670} C_VEL
LIN {X 0,Y 113.598,Z 857.696,A -85,B 0,C 180,E1 23685.46,E2 23685.46} C_VEL
LIN {X 0,Y 122.598,Z 850.019,A -85,B 0,C 180,E1 23703.762,E2 23703.762} C_VEL
LIN {X 0,Y 138.71,Z 837.952,A -85,B 0,C 180,E1 23717.458,E2 23717.458} C_VEL
LIN {X 0,Y 162.281,Z 818.463,A -85,B 0,C 180,E1 23728.554,E2 23728.554} C_VEL
LIN {X 0,Y 185.342,Z 795.926,A -85,B 0,C 180,E1 23735.415,E2 23735.415} C_VEL
LIN {X 0,Y 205.303,Z 772.149,A -85,B 0,C 180,E1 23739.716,E2 23739.716} C_VEL
LIN {X 0,Y 207.072,Z 763.292,A -85,B 0,C 180,E1 23744.74,E2 23744.74} C_VEL
LIN {X 0,Y 208.016,Z 755.004,A -85,B 0,C 180,E1 23751.638,E2 23751.638} C_VEL
LIN {X 0,Y 208.512,Z 751.669,A -85,B 0,C 180,E1 23755.844,E2 23755.844} C_VEL
LIN {X 0,Y 208.785,Z 750.071,A -85,B 0,C 180,E1 23760.008,E2 23760.008} C_VEL
LIN {X 0,Y 207.608,Z 752.736,A -85,B 0,C 180,E1 23766.288,E2 23766.288} C_VEL
LIN {X 0,Y 205.854,Z 760.106,A -85,B 0,C 180,E1 23773.809,E2 23773.809} C_VEL
LIN {X 0,Y 210.136,Z 783.049,A -85,B 0,C 180,E1 23792.783,E2 23792.783} C_VEL
LIN {X 0,Y 222.818,Z 796.529,A -85,B 0,C 180,E1 23804.292,E2 23804.292} C_VEL
LIN {X 0,Y 234.539,Z 808.628,A -85,B 0,C 180,E1 23813.119,E2 23813.119} C_VEL
LIN {X 0,Y 242.967,Z 817.073,A -85,B 0,C 180,E1 23820.098,E2 23820.098} C_VEL
LIN {X 0,Y 250.269,Z 824.076,A -85,B 0,C 180,E1 23827.343,E2 23827.343} C_VEL
LIN {X 0,Y 255.492,Z 829.265,A -85,B 0,C 180,E1 23834.534,E2 23834.534} C_VEL
LIN {X 0,Y 260.132,Z 832.004,A -85,B 0,C 180,E1 23841.699,E2 23841.699} C_VEL
LIN {X 0,Y 261.794,Z 832.779,A -85,B 0,C 180,E1 23846.684,E2 23846.684} C_VEL
LIN {X 0,Y 261.706,Z 832.854,A -85,B 0,C 180,E1 23853.317,E2 23853.317} C_VEL
LIN {X 0,Y 260.175,Z 831.904,A -85,B 0,C 180,E1 23858.367,E2 23858.367} C_VEL
LIN {X 0,Y 255.206,Z 829.036,A -85,B 0,C 180,E1 23865.713,E2 23865.713} C_VEL
LIN {X 0,Y 251.049,Z 828.454,A -85,B 0,C 180,E1 23868.523,E2 23868.523} C_VEL
LIN {X 0,Y 242.488,Z 826.705,A -85,B 0,C 180,E1 23873.254,E2 23873.254} C_VEL
LIN {X 0,Y 235.849,Z 820.346,A -85,B 0,C 180,E1 23879.859,E2 23879.859} C_VEL
LIN {X 0,Y 226.765,Z 811.118,A -85,B 0,C 180,E1 23887.405,E2 23887.405} C_VEL
LIN {X 0,Y 214.786,Z 799.478,A -85,B 0,C 180,E1 23896.576,E2 23896.576} C_VEL
LIN {X 0,Y 200.009,Z 780.502,A -85,B 0,C 180,E1 23914.266,E2 23914.266} C_VEL
LIN {X 0,Y 201.783,Z 761.811,A -85,B 0,C 180,E1 23930.272,E2 23930.272} C_VEL
LIN {X 0,Y 203.117,Z 757.776,A -85,B 0,C 180,E1 23935.718,E2 23935.718} C_VEL
LIN {X 0,Y 203.989,Z 756.408,A -85,B 0,C 180,E1 23939.992,E2 23939.992} C_VEL
LIN {X 0,Y 203.228,Z 759.613,A -85,B 0,C 180,E1 23946.408,E2 23946.408} C_VEL
LIN {X 0,Y 202.147,Z 766.657,A -85,B 0,C 180,E1 23953.174,E2 23953.174} C_VEL
LIN {X 0,Y 200.375,Z 774.261,A -85,B 0,C 180,E1 23958.116,E2 23958.116} C_VEL
LIN {X 0,Y 197.79,Z 778.148,A -85,B 0,C 180,E1 23959.045,E2 23959.045} C_VEL
LIN {X 0,Y 172.768,Z 805.07,A -85,B 0,C 180,E1 23964.603,E2 23964.603} C_VEL
LIN {X 0,Y 148.317,Z 826.332,A -85,B 0,C 180,E1 23972.629,E2 23972.629} C_VEL
LIN {X 0,Y 125.349,Z 843.389,A -85,B 0,C 180,E1 23985.326,E2 23985.326} C_VEL
LIN {X 0,Y 109.738,Z 854.244,A -85,B 0,C 180,E1 24003.122,E2 24003.122} C_VEL
LIN {X 0,Y 104.597,Z 858.857,A -85,B 0,C 180,E1 24021.677,E2 24021.677} C_VEL
LIN {X 0,Y 104.696,Z 859.336,A -85,B 0,C 180,E1 24030,E2 24030} C_VEL
LIN {X 0,Y 105.913,Z 857.459,A -85,B 0,C 180,E1 24046.613,E2 24046.613} C_VEL
LIN {X 0,Y 115.949,Z 849.78,A -85,B 0,C 180,E1 24065.987,E2 24065.987} C_VEL
LIN {X 0,Y 133.36,Z 837.712,A -85,B 0,C 180,E1 24080.026,E2 24080.026} C_VEL
LIN {X 0,Y 158.789,Z 817.75,A -85,B 0,C 180,E1 24091.247,E2 24091.247} C_VEL
LIN {X 0,Y 183.171,Z 794.585,A -85,B 0,C 180,E1 24097.953,E2 24097.953} C_VEL
LIN {X 0,Y 199.358,Z 776.185,A -85,B 0,C 180,E1 24101.239,E2 24101.239} C_VEL
LIN {X 0,Y 201.133,Z 771.285,A -85,B 0,C 180,E1 24103.613,E2 24103.613} C_VEL
LIN {X 0,Y 202.827,Z 762.474,A -85,B 0,C 180,E1 24110.326,E2 24110.326} C_VEL
LIN {X 0,Y 203.551,Z 758.1,A -85,B 0,C 180,E1 24115.742,E2 24115.742} C_VEL
LIN {X 0,Y 203.986,Z 756.411,A -85,B 0,C 180,E1 24120.008,E2 24120.008} C_VEL
LIN {X 0,Y 202.545,Z 759.17,A -85,B 0,C 180,E1 24126.446,E2 24126.446} C_VEL
LIN {X 0,Y 200.696,Z 765.478,A -85,B 0,C 180,E1 24133.088,E2 24133.088} C_VEL
LIN {X 0,Y 203.77,Z 787.698,A -85,B 0,C 180,E1 24152.602,E2 24152.602} C_VEL
LIN {X 0,Y 216.135,Z 800.667,A -85,B 0,C 180,E1 24164.476,E2 24164.476} C_VEL
LIN {X 0,Y 228.324,Z 813.044,A -85,B 0,C 180,E1 24173.971,E2 24173.971} C_VEL
LIN {X 0,Y 235.761,Z 820.332,A -85,B 0,C 180,E1 24180.142,E2 24180.142} C_VEL
LIN {X 0,Y 242.573,Z 826.841,A -85,B 0,C 180,E1 24186.855,E2 24186.855} C_VEL
LIN {X 0,Y 246.548,Z 830.978,A -85,B 0,C 180,E1 24192.118,E2 24192.118} C_VEL
LIN {X 0,Y 251.757,Z 834.618,A -85,B 0,C 180,E1 24199.606,E2 24199.606} C_VEL
LIN {X 0,Y 253.571,Z 835.463,A -85,B 0,C 180,E1 24203.141,E2 24203.141} C_VEL
LIN {X 0,Y 254.547,Z 836.023,A -85,B 0,C 180,E1 24206.59,E2 24206.59} C_VEL
LIN {X 0,Y 254.491,Z 836.079,A -85,B 0,C 180,E1 24213.411,E2 24213.411} C_VEL
LIN {X 0,Y 253.69,Z 835.483,A -85,B 0,C 180,E1 24216.855,E2 24216.855} C_VEL
LIN {X 0,Y 249.445,Z 833.299,A -85,B 0,C 180,E1 24223.779,E2 24223.779} C_VEL
LIN {X 0,Y 243.608,Z 827.932,A -85,B 0,C 180,E1 24231.895,E2 24231.895} C_VEL
LIN {X 0,Y 242.488,Z 826.705,A -85,B 0,C 180,E1 24233.254,E2 24233.254} C_VEL
LIN {X 0,Y 237.387,Z 825.127,A -85,B 0,C 180,E1 24236.116,E2 24236.116} C_VEL
LIN {X 0,Y 227.168,Z 822.03,A -85,B 0,C 180,E1 24240.92,E2 24240.92} C_VEL
LIN {X 0,Y 217.465,Z 812.352,A -85,B 0,C 180,E1 24248.8,E2 24248.8} C_VEL
LIN {X 0,Y 205.72,Z 801.209,A -85,B 0,C 180,E1 24258.51,E2 24258.51} C_VEL
LIN {X 0,Y 193.452,Z 777.737,A -85,B 0,C 180,E1 24281.748,E2 24281.748} C_VEL
LIN {X 0,Y 196.698,Z 767.2,A -85,B 0,C 180,E1 24291.137,E2 24291.137} C_VEL
LIN {X 0,Y 198.039,Z 764.121,A -85,B 0,C 180,E1 24295.608,E2 24295.608} C_VEL
LIN {X 0,Y 199.025,Z 762.637,A -85,B 0,C 180,E1 24299.992,E2 24299.992} C_VEL
LIN {X 0,Y 198.105,Z 765.961,A -85,B 0,C 180,E1 24306.511,E2 24306.511} C_VEL
LIN {X 0,Y 196.396,Z 773.052,A -85,B 0,C 180,E1 24313.363,E2 24313.363} C_VEL
LIN {X 0,Y 195.112,Z 777.825,A -85,B 0,C 180,E1 24316.556,E2 24316.556} C_VEL
LIN {X 0,Y 172.735,Z 801.827,A -85,B 0,C 180,E1 24321.362,E2 24321.362} C_VEL
LIN {X 0,Y 146.96,Z 824.024,A -85,B 0,C 180,E1 24328.871,E2 24328.871} C_VEL
LIN {X 0,Y 123.564,Z 840.544,A -85,B 0,C 180,E1 24340.02,E2 24340.02} C_VEL
LIN {X 0,Y 106.384,Z 851.612,A -85,B 0,C 180,E1 24355.3,E2 24355.3} C_VEL
LIN {X 0,Y 98.259,Z 857.223,A -85,B 0,C 180,E1 24372.051,E2 24372.051} C_VEL
LIN {X 0,Y 96.775,Z 859.102,A -85,B 0,C 180,E1 24390,E2 24390} C_VEL
LIN {X 0,Y 98.262,Z 857.223,A -85,B 0,C 180,E1 24407.949,E2 24407.949} C_VEL
LIN {X 0,Y 109.522,Z 849.541,A -85,B 0,C 180,E1 24428.469,E2 24428.469} C_VEL
LIN {X 0,Y 128.297,Z 837.472,A -85,B 0,C 180,E1 24442.805,E2 24442.805} C_VEL
LIN {X 0,Y 155.067,Z 817.511,A -85,B 0,C 180,E1 24453.863,E2 24453.863} C_VEL
LIN {X 0,Y 179.7,Z 794.975,A -85,B 0,C 180,E1 24460.196,E2 24460.196} C_VEL
LIN {X 0,Y 195.151,Z 777.817,A -85,B 0,C 180,E1 24463.416,E2 24463.416} C_VEL
LIN {X 0,Y 197.331,Z 769.258,A -85,B 0,C 180,E1 24469.785,E2 24469.785} C_VEL
LIN {X 0,Y 198.503,Z 764.443,A -85,B 0,C 180,E1 24475.634,E2 24475.634} C_VEL
LIN {X 0,Y 199.028,Z 762.633,A -85,B 0,C 180,E1 24480.008,E2 24480.008} C_VEL
LIN {X 0,Y 197.349,Z 765.523,A -85,B 0,C 180,E1 24486.614,E2 24486.614} C_VEL
LIN {X 0,Y 194.917,Z 772.122,A -85,B 0,C 180,E1 24493.483,E2 24493.483} C_VEL
LIN {X 0,Y 198.774,Z 794.015,A -85,B 0,C 180,E1 24514.287,E2 24514.287} C_VEL
LIN {X 0,Y 210.889,Z 806.026,A -85,B 0,C 180,E1 24525.893,E2 24525.893} C_VEL
LIN {X 0,Y 222.028,Z 817.15,A -85,B 0,C 180,E1 24534.925,E2 24534.925} C_VEL
LIN {X 0,Y 229.912,Z 824.895,A -85,B 0,C 180,E1 24541.659,E2 24541.659} C_VEL
LIN {X 0,Y 236.429,Z 830.998,A -85,B 0,C 180,E1 24548.359,E2 24548.359} C_VEL
LIN {X 0,Y 241.503,Z 835.885,A -85,B 0,C 180,E1 24555.477,E2 24555.477} C_VEL
LIN {X 0,Y 245.141,Z 838.002,A -85,B 0,C 180,E1 24561.217,E2 24561.217} C_VEL
LIN {X 0,Y 247.166,Z 838.983,A -85,B 0,C 180,E1 24566.488,E2 24566.488} C_VEL
LIN {X 0,Y 247.121,Z 839.034,A -85,B 0,C 180,E1 24573.513,E2 24573.513} C_VEL
LIN {X 0,Y 245.171,Z 837.936,A -85,B 0,C 180,E1 24578.828,E2 24578.828} C_VEL
LIN {X 0,Y 240.216,Z 834.9,A -85,B 0,C 180,E1 24586.297,E2 24586.297} C_VEL
LIN {X 0,Y 235.253,Z 829.826,A -85,B 0,C 180,E1 24593.004,E2 24593.004} C_VEL
LIN {X 0,Y 227.925,Z 822.771,A -85,B 0,C 180,E1 24600.272,E2 24600.272} C_VEL
LIN {X 0,Y 227.168,Z 822.03,A -85,B 0,C 180,E1 24600.92,E2 24600.92} C_VEL
LIN {X 0,Y 221.301,Z 819.454,A -85,B 0,C 180,E1 24603.845,E2 24603.845} C_VEL
LIN {X 0,Y 209.985,Z 815.337,A -85,B 0,C 180,E1 24608.815,E2 24608.815} C_VEL
LIN {X 0,Y 197.946,Z 804.336,A -85,B 0,C 180,E1 24619.328,E2 24619.328} C_VEL
LIN {X 0,Y 187.65,Z 782.665,A -85,B 0,C 180,E1 24642.381,E2 24642.381} C_VEL
LIN {X 0,Y 191.426,Z 772.685,A -85,B 0,C 180,E1 24651.909,E2 24651.909} C_VEL
LIN {X 0,Y 192.642,Z 770.211,A -85,B 0,C 180,E1 24655.484,E2 24655.484} C_VEL
LIN {X 0,Y 193.815,Z 768.674,A -85,B 0,C 180,E1 24659.992,E2 24659.992} C_VEL
LIN {X 0,Y 192.643,Z 772.1,A -85,B 0,C 180,E1 24666.697,E2 24666.697} C_VEL
LIN {X 0,Y 190.94,Z 778.079,A -85,B 0,C 180,E1 24672.586,E2 24672.586} C_VEL
LIN {X 0,Y 189.821,Z 781.12,A -85,B 0,C 180,E1 24674.828,E2 24674.828} C_VEL
LIN {X 0,Y 163.453,Z 807.547,A -85,B 0,C 180,E1 24680.303,E2 24680.303} C_VEL
LIN {X 0,Y 135.226,Z 829.425,A -85,B 0,C 180,E1 24688.933,E2 24688.933} C_VEL
LIN {X 0,Y 111.459,Z 844.565,A -85,B 0,C 180,E1 24701.665,E2 24701.665} C_VEL
LIN {X 0,Y 94.282,Z 854.654,A -85,B 0,C 180,E1 24721.2,E2 24721.2} C_VEL
LIN {X 0,Y 88.888,Z 858.387,A -85,B 0,C 180,E1 24740.193,E2 24740.193} C_VEL
LIN {X 0,Y 88.874,Z 858.869,A -85,B 0,C 180,E1 24750,E2 24750} C_VEL
LIN {X 0,Y 90.696,Z 856.987,A -85,B 0,C 180,E1 24769.504,E2 24769.504} C_VEL
LIN {X 0,Y 103.304,Z 849.302,A -85,B 0,C 180,E1 24791.265,E2 24791.265} C_VEL
LIN {X 0,Y 123.57,Z 837.233,A -85,B 0,C 180,E1 24805.797,E2 24805.797} C_VEL
LIN {X 0,Y 150.637,Z 818.061,A -85,B 0,C 180,E1 24816.307,E2 24816.307} C_VEL
LIN {X 0,Y 176.649,Z 795.233,A -85,B 0,C 180,E1 24822.547,E2 24822.547} C_VEL
LIN {X 0,Y 189.47,Z 781.75,A -85,B 0,C 180,E1 24824.859,E2 24824.859} C_VEL
LIN {X 0,Y 192.108,Z 774.13,A -85,B 0,C 180,E1 24830.94,E2 24830.94} C_VEL
LIN {X 0,Y 193.128,Z 770.539,A -85,B 0,C 180,E1 24835.512,E2 24835.512} C_VEL
LIN {X 0,Y 193.83,Z 768.657,A -85,B 0,C 180,E1 24840.008,E2 24840.008} C_VEL
LIN {X 0,Y 191.864,Z 771.701,A -85,B 0,C 180,E1 24846.806,E2 24846.806} C_VEL
LIN {X 0,Y 188.898,Z 778.543,A -85,B 0,C 180,E1 24853.921,E2 24853.921} C_VEL
LIN {X 0,Y 193.64,Z 799.857,A -85,B 0,C 180,E1 24875.912,E2 24875.912} C_VEL
LIN {X 0,Y 205.543,Z 811.217,A -85,B 0,C 180,E1 24887.452,E2 24887.452} C_VEL
LIN {X 0,Y 216.903,Z 822.132,A -85,B 0,C 180,E1 24896.901,E2 24896.901} C_VEL
LIN {X 0,Y 224.902,Z 829.941,A -85,B 0,C 180,E1 24904.171,E2 24904.171} C_VEL
LIN {X 0,Y 230.687,Z 835.457,A -85,B 0,C 180,E1 24910.843,E2 24910.843} C_VEL
LIN {X 0,Y 236.266,Z 839.889,A -85,B 0,C 180,E1 24918.916,E2 24918.916} C_VEL
LIN {X 0,Y 238.451,Z 840.968,A -85,B 0,C 180,E1 24922.704,E2 24922.704} C_VEL
LIN {X 0,Y 239.645,Z 841.607,A -85,B 0,C 180,E1 24926.378,E2 24926.378} C_VEL
LIN {X 0,Y 239.959,Z 841.836,A -85,B 0,C 180,E1 24930,E2 24930} C_VEL
LIN {X 0,Y 239.613,Z 841.658,A -85,B 0,C 180,E1 24933.623,E2 24933.623} C_VEL
LIN {X 0,Y 238.568,Z 840.998,A -85,B 0,C 180,E1 24937.292,E2 24937.292} C_VEL
LIN {X 0,Y 233.574,Z 838.128,A -85,B 0,C 180,E1 24945.028,E2 24945.028} C_VEL
LIN {X 0,Y 228.621,Z 833.296,A -85,B 0,C 180,E1 24951.991,E2 24951.991} C_VEL
LIN {X 0,Y 221.252,Z 826.173,A -85,B 0,C 180,E1 24959.436,E2 24959.436} C_VEL
LIN {X 0,Y 211.13,Z 816.39,A -85,B 0,C 180,E1 24967.914,E2 24967.914} C_VEL
LIN {X 0,Y 209.985,Z 815.337,A -85,B 0,C 180,E1 24968.815,E2 24968.815} C_VEL
LIN {X 0,Y 203.87,Z 812.877,A -85,B 0,C 180,E1 24971.956,E2 24971.956} C_VEL
LIN {X 0,Y 192.829,Z 809.822,A -85,B 0,C 180,E1 24977.441,E2 24977.441} C_VEL
LIN {X 0,Y 181.555,Z 788.116,A -85,B 0,C 180,E1 25002.333,E2 25002.333} C_VEL
LIN {X 0,Y 185.971,Z 778.169,A -85,B 0,C 180,E1 25012.382,E2 25012.382} C_VEL
LIN {X 0,Y 188.483,Z 774.623,A -85,B 0,C 180,E1 25019.992,E2 25019.992} C_VEL
LIN {X 0,Y 187.048,Z 778.206,A -85,B 0,C 180,E1 25026.965,E2 25026.965} C_VEL
LIN {X 0,Y 184.776,Z 784.155,A -85,B 0,C 180,E1 25032.757,E2 25032.757} C_VEL
LIN {X 0,Y 182.943,Z 786.508,A -85,B 0,C 180,E1 25033.482,E2 25033.482} C_VEL
LIN {X 0,Y 155.88,Z 811.307,A -85,B 0,C 180,E1 25038.736,E2 25038.736} C_VEL
LIN {X 0,Y 130.7,Z 829.734,A -85,B 0,C 180,E1 25046.133,E2 25046.133} C_VEL
LIN {X 0,Y 106.249,Z 844.323,A -85,B 0,C 180,E1 25058.394,E2 25058.394} C_VEL
LIN {X 0,Y 87.302,Z 854.416,A -85,B 0,C 180,E1 25078.649,E2 25078.649} C_VEL
LIN {X 0,Y 81.043,Z 858.151,A -85,B 0,C 180,E1 25099.233,E2 25099.233} C_VEL
LIN {X 0,Y 80.949,Z 858.635,A -85,B 0,C 180,E1 25110,E2 25110} C_VEL
LIN {X 0,Y 83.182,Z 856.75,A -85,B 0,C 180,E1 25131.348,E2 25131.348} C_VEL
LIN {X 0,Y 97.29,Z 849.1,A -85,B 0,C 180,E1 25154.339,E2 25154.339} C_VEL
LIN {X 0,Y 119.018,Z 837.111,A -85,B 0,C 180,E1 25168.92,E2 25168.92} C_VEL
LIN {X 0,Y 147.591,Z 817.824,A -85,B 0,C 180,E1 25179.164,E2 25179.164} C_VEL
LIN {X 0,Y 174.161,Z 795.237,A -85,B 0,C 180,E1 25185.024,E2 25185.024} C_VEL
LIN {X 0,Y 184.003,Z 785.353,A -85,B 0,C 180,E1 25186.683,E2 25186.683} C_VEL
LIN {X 0,Y 186.303,Z 780.25,A -85,B 0,C 180,E1 25190.655,E2 25190.655} C_VEL
LIN {X 0,Y 188.014,Z 775.524,A -85,B 0,C 180,E1 25197.701,E2 25197.701} C_VEL
LIN {X 0,Y 188.508,Z 774.595,A -85,B 0,C 180,E1 25200.008,E2 25200.008} C_VEL
LIN {X 0,Y 187.163,Z 776.217,A -85,B 0,C 180,E1 25204.648,E2 25204.648} C_VEL
LIN {X 0,Y 183.898,Z 782.133,A -85,B 0,C 180,E1 25211.884,E2 25211.884} C_VEL
LIN {X 0,Y 185.937,Z 803.097,A -85,B 0,C 180,E1 25234.759,E2 25234.759} C_VEL
LIN {X 0,Y 197.923,Z 814.175,A -85,B 0,C 180,E1 25247.217,E2 25247.217} C_VEL
LIN {X 0,Y 207.754,Z 823.131,A -85,B 0,C 180,E1 25255.714,E2 25255.714} C_VEL
LIN {X 0,Y 215.978,Z 830.955,A -85,B 0,C 180,E1 25262.98,E2 25262.98} C_VEL
LIN {X 0,Y 222.536,Z 837.139,A -85,B 0,C 180,E1 25270.112,E2 25270.112} C_VEL
LIN {X 0,Y 228.322,Z 842.014,A -85,B 0,C 180,E1 25278.525,E2 25278.525} C_VEL
LIN {X 0,Y 230.64,Z 843.2,A -85,B 0,C 180,E1 25282.456,E2 25282.456} C_VEL
LIN {X 0,Y 231.993,Z 843.834,A -85,B 0,C 180,E1 25286.258,E2 25286.258} C_VEL
LIN {X 0,Y 232.394,Z 844.07,A -85,B 0,C 180,E1 25290,E2 25290} C_VEL
LIN {X 0,Y 231.973,Z 843.88,A -85,B 0,C 180,E1 25293.742,E2 25293.742} C_VEL
LIN {X 0,Y 229.89,Z 842.858,A -85,B 0,C 180,E1 25298.893,E2 25298.893} C_VEL
LIN {X 0,Y 225.536,Z 839.991,A -85,B 0,C 180,E1 25305.577,E2 25305.577} C_VEL
LIN {X 0,Y 220.102,Z 834.75,A -85,B 0,C 180,E1 25312.89,E2 25312.89} C_VEL
LIN {X 0,Y 213.074,Z 828.006,A -85,B 0,C 180,E1 25319.828,E2 25319.828} C_VEL
LIN {X 0,Y 202.93,Z 818.639,A -85,B 0,C 180,E1 25328.424,E2 25328.424} C_VEL
LIN {X 0,Y 192.829,Z 809.822,A -85,B 0,C 180,E1 25337.441,E2 25337.441} C_VEL
LIN {X 0,Y 187.14,Z 807.973,A -85,B 0,C 180,E1 25340.973,E2 25340.973} C_VEL
LIN {X 0,Y 178.275,Z 806.226,A -85,B 0,C 180,E1 25346.537,E2 25346.537} C_VEL
LIN {X 0,Y 177.8,Z 805.751,A -85,B 0,C 180,E1 25347.213,E2 25347.213} C_VEL
LIN {X 0,Y 180.123,Z 783.952,A -85,B 0,C 180,E1 25372.349,E2 25372.349} C_VEL
LIN {X 0,Y 182.887,Z 780.313,A -85,B 0,C 180,E1 25379.991,E2 25379.991} C_VEL
LIN {X 0,Y 181.264,Z 783.881,A -85,B 0,C 180,E1 25386.944,E2 25386.944} C_VEL
LIN {X 0,Y 179.485,Z 787.978,A -85,B 0,C 180,E1 25391.137,E2 25391.137} C_VEL
LIN {X 0,Y 150.114,Z 813.733,A -85,B 0,C 180,E1 25396.63,E2 25396.63} C_VEL
LIN {X 0,Y 121.197,Z 833.192,A -85,B 0,C 180,E1 25405.082,E2 25405.082} C_VEL
LIN {X 0,Y 94.243,Z 847.702,A -85,B 0,C 180,E1 25419.964,E2 25419.964} C_VEL
LIN {X 0,Y 78.552,Z 855.045,A -85,B 0,C 180,E1 25439.392,E2 25439.392} C_VEL
LIN {X 0,Y 73.221,Z 857.915,A -85,B 0,C 180,E1 25458.067,E2 25458.067} C_VEL
LIN {X 0,Y 73.048,Z 858.401,A -85,B 0,C 180,E1 25470,E2 25470} C_VEL
LIN {X 0,Y 75.764,Z 856.513,A -85,B 0,C 180,E1 25493.558,E2 25493.558} C_VEL
LIN {X 0,Y 90.734,Z 849.31,A -85,B 0,C 180,E1 25516.996,E2 25516.996} C_VEL
LIN {X 0,Y 114.967,Z 836.919,A -85,B 0,C 180,E1 25532.336,E2 25532.336} C_VEL
LIN {X 0,Y 145.107,Z 817.45,A -85,B 0,C 180,E1 25542.196,E2 25542.196} C_VEL
LIN {X 0,Y 171.979,Z 795.271,A -85,B 0,C 180,E1 25547.56,E2 25547.56} C_VEL
LIN {X 0,Y 179.504,Z 787.963,A -85,B 0,C 180,E1 25548.861,E2 25548.861} C_VEL
LIN {X 0,Y 181.877,Z 782.379,A -85,B 0,C 180,E1 25555.234,E2 25555.234} C_VEL
LIN {X 0,Y 182.915,Z 780.285,A -85,B 0,C 180,E1 25560.009,E2 25560.009} C_VEL
LIN {X 0,Y 180.056,Z 784.085,A -85,B 0,C 180,E1 25567.855,E2 25567.855} C_VEL
LIN {X 0,Y 178.341,Z 806.226,A -85,B 0,C 180,E1 25593.499,E2 25593.499} C_VEL
LIN {X 0,Y 189.282,Z 816.306,A -85,B 0,C 180,E1 25606.056,E2 25606.056} C_VEL
LIN {X 0,Y 200.531,Z 825.903,A -85,B 0,C 180,E1 25616.163,E2 25616.163} C_VEL
LIN {X 0,Y 208.714,Z 833.306,A -85,B 0,C 180,E1 25623.526,E2 25623.526} C_VEL
LIN {X 0,Y 214.173,Z 838.403,A -85,B 0,C 180,E1 25629.301,E2 25629.301} C_VEL
LIN {X 0,Y 220.291,Z 843.759,A -85,B 0,C 180,E1 25638.101,E2 25638.101} C_VEL
LIN {X 0,Y 222.724,Z 845.039,A -85,B 0,C 180,E1 25642.186,E2 25642.186} C_VEL
LIN {X 0,Y 224.256,Z 845.757,A -85,B 0,C 180,E1 25646.129,E2 25646.129} C_VEL
LIN {X 0,Y 224.754,Z 846.011,A -85,B 0,C 180,E1 25650,E2 25650} C_VEL
LIN {X 0,Y 224.249,Z 845.8,A -85,B 0,C 180,E1 25653.871,E2 25653.871} C_VEL
LIN {X 0,Y 222.822,Z 845.036,A -85,B 0,C 180,E1 25657.811,E2 25657.811} C_VEL
LIN {X 0,Y 217.348,Z 841.548,A -85,B 0,C 180,E1 25666.179,E2 25666.179} C_VEL
LIN {X 0,Y 212.803,Z 837.036,A -85,B 0,C 180,E1 25672.329,E2 25672.329} C_VEL
LIN {X 0,Y 204.846,Z 829.567,A -85,B 0,C 180,E1 25680.164,E2 25680.164} C_VEL
LIN {X 0,Y 194.755,Z 820.851,A -85,B 0,C 180,E1 25688.965,E2 25688.965} C_VEL
LIN {X 0,Y 184.293,Z 812.171,A -85,B 0,C 180,E1 25698.901,E2 25698.901} C_VEL
LIN {X 0,Y 177.8,Z 805.751,A -85,B 0,C 180,E1 25707.213,E2 25707.213} C_VEL
LIN {X 0,Y 172.272,Z 803.788,A -85,B 0,C 180,E1 25712.63,E2 25712.63} C_VEL
LIN {X 0,Y 168.402,Z 801.602,A -85,B 0,C 180,E1 25718.332,E2 25718.332} C_VEL
LIN {X 0,Y 174.173,Z 789.303,A -85,B 0,C 180,E1 25732.611,E2 25732.611} C_VEL
LIN {X 0,Y 177.202,Z 785.931,A -85,B 0,C 180,E1 25739.991,E2 25739.991} C_VEL
LIN {X 0,Y 175.135,Z 789.725,A -85,B 0,C 180,E1 25747.291,E2 25747.291} C_VEL
LIN {X 0,Y 173.256,Z 792.365,A -85,B 0,C 180,E1 25749.39,E2 25749.39} C_VEL
LIN {X 0,Y 144.562,Z 816.036,A -85,B 0,C 180,E1 25754.354,E2 25754.354} C_VEL
LIN {X 0,Y 112.458,Z 836.105,A -85,B 0,C 180,E1 25763.559,E2 25763.559} C_VEL
LIN {X 0,Y 85.092,Z 849.218,A -85,B 0,C 180,E1 25779.329,E2 25779.329} C_VEL
LIN {X 0,Y 68.468,Z 856.275,A -85,B 0,C 180,E1 25803.752,E2 25803.752} C_VEL
LIN {X 0,Y 65.118,Z 858.167,A -85,B 0,C 180,E1 25830,E2 25830} C_VEL
LIN {X 0,Y 68.47,Z 856.275,A -85,B 0,C 180,E1 25856.248,E2 25856.248} C_VEL
LIN {X 0,Y 85.081,Z 849.22,A -85,B 0,C 180,E1 25880.67,E2 25880.67} C_VEL
LIN {X 0,Y 112.451,Z 836.112,A -85,B 0,C 180,E1 25896.432,E2 25896.432} C_VEL
LIN {X 0,Y 144.551,Z 816.034,A -85,B 0,C 180,E1 25905.664,E2 25905.664} C_VEL
LIN {X 0,Y 173.259,Z 792.368,A -85,B 0,C 180,E1 25910.599,E2 25910.599} C_VEL
LIN {X 0,Y 174.848,Z 790.292,A -85,B 0,C 180,E1 25912.002,E2 25912.002} C_VEL
LIN {X 0,Y 176.575,Z 786.958,A -85,B 0,C 180,E1 25917.306,E2 25917.306} C_VEL
LIN {X 0,Y 177.228,Z 785.906,A -85,B 0,C 180,E1 25920.009,E2 25920.009} C_VEL
LIN {X 0,Y 174.148,Z 789.355,A -85,B 0,C 180,E1 25927.502,E2 25927.502} C_VEL
LIN {X 0,Y 170.792,Z 809.279,A -85,B 0,C 180,E1 25952.143,E2 25952.143} C_VEL
LIN {X 0,Y 182.075,Z 819.566,A -85,B 0,C 180,E1 25966.251,E2 25966.251} C_VEL
LIN {X 0,Y 193.431,Z 828.704,A -85,B 0,C 180,E1 25976.776,E2 25976.776} C_VEL
LIN {X 0,Y 201.591,Z 835.656,A -85,B 0,C 180,E1 25984.338,E2 25984.338} C_VEL
LIN {X 0,Y 207.788,Z 841.394,A -85,B 0,C 180,E1 25991.324,E2 25991.324} C_VEL
LIN {X 0,Y 212.108,Z 845.062,A -85,B 0,C 180,E1 25997.635,E2 25997.635} C_VEL
LIN {X 0,Y 214.675,Z 846.591,A -85,B 0,C 180,E1 26001.891,E2 26001.891} C_VEL
LIN {X 0,Y 216.41,Z 847.389,A -85,B 0,C 180,E1 26005.988,E2 26005.988} C_VEL
LIN {X 0,Y 217.031,Z 847.662,A -85,B 0,C 180,E1 26010,E2 26010} C_VEL
LIN {X 0,Y 216.414,Z 847.433,A -85,B 0,C 180,E1 26014.012,E2 26014.012} C_VEL
LIN {X 0,Y 214.404,Z 846.421,A -85,B 0,C 180,E1 26018.613,E2 26018.613} C_VEL
LIN {X 0,Y 209.021,Z 842.658,A -85,B 0,C 180,E1 26026.842,E2 26026.842} C_VEL
LIN {X 0,Y 204.017,Z 837.66,A -85,B 0,C 180,E1 26033.346,E2 26033.346} C_VEL
LIN {X 0,Y 195.412,Z 830.204,A -85,B 0,C 180,E1 26041.528,E2 26041.528} C_VEL
LIN {X 0,Y 185.068,Z 821.926,A -85,B 0,C 180,E1 26050.88,E2 26050.88} C_VEL
LIN {X 0,Y 174.124,Z 813.069,A -85,B 0,C 180,E1 26062.497,E2 26062.497} C_VEL
LIN {X 0,Y 168.402,Z 801.602,A -85,B 0,C 180,E1 26078.332,E2 26078.332} C_VEL
LIN {X 0,Y 166.392,Z 799.273,A -85,B 0,C 180,E1 26084.249,E2 26084.249} C_VEL
LIN {X 0,Y 166.305,Z 796.773,A -85,B 0,C 180,E1 26090.218,E2 26090.218} C_VEL
LIN {X 0,Y 169.138,Z 793.291,A -85,B 0,C 180,E1 26094.855,E2 26094.855} C_VEL
LIN {X 0,Y 171.211,Z 791.296,A -85,B 0,C 180,E1 26099.991,E2 26099.991} C_VEL
LIN {X 0,Y 169.152,Z 794.766,A -85,B 0,C 180,E1 26106.831,E2 26106.831} C_VEL
LIN {X 0,Y 141.013,Z 816.974,A -85,B 0,C 180,E1 26111.55,E2 26111.55} C_VEL
LIN {X 0,Y 109.805,Z 835.676,A -85,B 0,C 180,E1 26119.534,E2 26119.534} C_VEL
LIN {X 0,Y 81.445,Z 848.485,A -85,B 0,C 180,E1 26133.872,E2 26133.872} C_VEL
LIN {X 0,Y 61.36,Z 856.037,A -85,B 0,C 180,E1 26160.43,E2 26160.43} C_VEL
LIN {X 0,Y 57.2,Z 857.933,A -85,B 0,C 180,E1 26190,E2 26190} C_VEL
LIN {X 0,Y 61.368,Z 856.038,A -85,B 0,C 180,E1 26219.567,E2 26219.567} C_VEL
LIN {X 0,Y 81.387,Z 848.503,A -85,B 0,C 180,E1 26246.101,E2 26246.101} C_VEL
LIN {X 0,Y 109.464,Z 835.871,A -85,B 0,C 180,E1 26260.326,E2 26260.326} C_VEL
LIN {X 0,Y 142.766,Z 815.796,A -85,B 0,C 180,E1 26268.807,E2 26268.807} C_VEL
LIN {X 0,Y 169.164,Z 794.756,A -85,B 0,C 180,E1 26273.169,E2 26273.169} C_VEL
LIN {X 0,Y 171.237,Z 791.272,A -85,B 0,C 180,E1 26280.009,E2 26280.009} C_VEL
LIN {X 0,Y 167.963,Z 794.775,A -85,B 0,C 180,E1 26287.449,E2 26287.449} C_VEL
LIN {X 0,Y 164.623,Z 814.041,A -85,B 0,C 180,E1 26313.502,E2 26313.502} C_VEL
LIN {X 0,Y 175.878,Z 823.489,A -85,B 0,C 180,E1 26327.523,E2 26327.523} C_VEL
LIN {X 0,Y 185.874,Z 831.005,A -85,B 0,C 180,E1 26337.064,E2 26337.064} C_VEL
LIN {X 0,Y 194.631,Z 837.895,A -85,B 0,C 180,E1 26345.372,E2 26345.372} C_VEL
LIN {X 0,Y 200.607,Z 843.296,A -85,B 0,C 180,E1 26352.429,E2 26352.429} C_VEL
LIN {X 0,Y 203.821,Z 845.988,A -85,B 0,C 180,E1 26357.123,E2 26357.123} C_VEL
LIN {X 0,Y 206.556,Z 847.75,A -85,B 0,C 180,E1 26361.57,E2 26361.57} C_VEL
LIN {X 0,Y 208.455,Z 848.627,A -85,B 0,C 180,E1 26365.835,E2 26365.835} C_VEL
LIN {X 0,Y 209.228,Z 848.916,A -85,B 0,C 180,E1 26370,E2 26370} C_VEL
LIN {X 0,Y 208.468,Z 848.673,A -85,B 0,C 180,E1 26374.165,E2 26374.165} C_VEL
LIN {X 0,Y 206.605,Z 847.719,A -85,B 0,C 180,E1 26378.428,E2 26378.428} C_VEL
LIN {X 0,Y 201.891,Z 844.512,A -85,B 0,C 180,E1 26385.661,E2 26385.661} C_VEL
LIN {X 0,Y 196.678,Z 839.516,A -85,B 0,C 180,E1 26392.638,E2 26392.638} C_VEL
LIN {X 0,Y 187.902,Z 832.483,A -85,B 0,C 180,E1 26401.178,E2 26401.178} C_VEL
LIN {X 0,Y 178.24,Z 825.24,A -85,B 0,C 180,E1 26410.126,E2 26410.126} C_VEL
LIN {X 0,Y 166.202,Z 815.87,A -85,B 0,C 180,E1 26423.685,E2 26423.685} C_VEL
LIN {X 0,Y 165.788,Z 797.43,A -85,B 0,C 180,E1 26449.467,E2 26449.467} C_VEL
LIN {X 0,Y 166.305,Z 796.773,A -85,B 0,C 180,E1 26450.218,E2 26450.218} C_VEL
LIN {X 0,Y 167.064,Z 795.178,A -85,B 0,C 180,E1 26454.677,E2 26454.677} C_VEL
LIN {X 0,Y 164.505,Z 797.446,A -85,B 0,C 180,E1 26462.463,E2 26462.463} C_VEL
LIN {X 0,Y 164.002,Z 798.156,A -85,B 0,C 180,E1 26463.961,E2 26463.961} C_VEL
LIN {X 0,Y 162.165,Z 799.885,A -85,B 0,C 180,E1 26465.096,E2 26465.096} C_VEL
LIN {X 0,Y 131.597,Z 821.984,A -85,B 0,C 180,E1 26469.716,E2 26469.716} C_VEL
LIN {X 0,Y 98.901,Z 839.398,A -85,B 0,C 180,E1 26478.285,E2 26478.285} C_VEL
LIN {X 0,Y 71.996,Z 850.178,A -85,B 0,C 180,E1 26492.734,E2 26492.734} C_VEL
LIN {X 0,Y 54.456,Z 855.827,A -85,B 0,C 180,E1 26516.466,E2 26516.466} C_VEL
LIN {X 0,Y 49.263,Z 857.698,A -85,B 0,C 180,E1 26550,E2 26550} C_VEL
LIN {X 0,Y 54.533,Z 855.8,A -85,B 0,C 180,E1 26583.73,E2 26583.73} C_VEL
LIN {X 0,Y 77.158,Z 848.263,A -85,B 0,C 180,E1 26611.106,E2 26611.106} C_VEL
LIN {X 0,Y 107.321,Z 835.467,A -85,B 0,C 180,E1 26624.51,E2 26624.51} C_VEL
LIN {X 0,Y 141.415,Z 815.56,A -85,B 0,C 180,E1 26632.034,E2 26632.034} C_VEL
LIN {X 0,Y 162.156,Z 799.898,A -85,B 0,C 180,E1 26634.885,E2 26634.885} C_VEL
LIN {X 0,Y 163.994,Z 798.162,A -85,B 0,C 180,E1 26636.039,E2 26636.039} C_VEL
LIN {X 0,Y 165.184,Z 796.569,A -85,B 0,C 180,E1 26640.01,E2 26640.01} C_VEL
LIN {X 0,Y 161.154,Z 800.288,A -85,B 0,C 180,E1 26647.765,E2 26647.765} C_VEL
LIN {X 0,Y 158.434,Z 818.596,A -85,B 0,C 180,E1 26674.997,E2 26674.997} C_VEL
LIN {X 0,Y 168.719,Z 826.521,A -85,B 0,C 180,E1 26687.992,E2 26687.992} C_VEL
LIN {X 0,Y 178.828,Z 833.6,A -85,B 0,C 180,E1 26697.863,E2 26697.863} C_VEL
LIN {X 0,Y 187.375,Z 839.815,A -85,B 0,C 180,E1 26706.17,E2 26706.17} C_VEL
LIN {X 0,Y 193.304,Z 844.776,A -85,B 0,C 180,E1 26713.46,E2 26713.46} C_VEL
LIN {X 0,Y 198.808,Z 848.711,A -85,B 0,C 180,E1 26721.944,E2 26721.944} C_VEL
LIN {X 0,Y 200.442,Z 849.514,A -85,B 0,C 180,E1 26725.668,E2 26725.668} C_VEL
LIN {X 0,Y 201.378,Z 849.831,A -85,B 0,C 180,E1 26730,E2 26730} C_VEL
LIN {X 0,Y 200.459,Z 849.562,A -85,B 0,C 180,E1 26734.332,E2 26734.332} C_VEL
LIN {X 0,Y 198.345,Z 848.492,A -85,B 0,C 180,E1 26738.782,E2 26738.782} C_VEL
LIN {X 0,Y 193.302,Z 844.783,A -85,B 0,C 180,E1 26746.53,E2 26746.53} C_VEL
LIN {X 0,Y 187.477,Z 839.812,A -85,B 0,C 180,E1 26753.816,E2 26753.816} C_VEL
LIN {X 0,Y 178.897,Z 833.55,A -85,B 0,C 180,E1 26762.173,E2 26762.173} C_VEL
LIN {X 0,Y 168.666,Z 826.502,A -85,B 0,C 180,E1 26772.045,E2 26772.045} C_VEL
LIN {X 0,Y 155.845,Z 815.105,A -85,B 0,C 180,E1 26790.969,E2 26790.969} C_VEL
LIN {X 0,Y 162.696,Z 798.662,A -85,B 0,C 180,E1 26814.651,E2 26814.651} C_VEL
LIN {X 0,Y 165.134,Z 796.609,A -85,B 0,C 180,E1 26819.99,E2 26819.99} C_VEL
LIN {X 0,Y 164.505,Z 797.446,A -85,B 0,C 180,E1 26822.463,E2 26822.463} C_VEL
LIN {X 0,Y 161.365,Z 800.21,A -85,B 0,C 180,E1 26823.763,E2 26823.763} C_VEL
LIN {X 0,Y 145.938,Z 811.562,A -85,B 0,C 180,E1 26824.018,E2 26824.018} C_VEL
LIN {X 0,Y 114.979,Z 830.456,A -85,B 0,C 180,E1 26829.032,E2 26829.032} C_VEL
LIN {X 0,Y 80.462,Z 845.676,A -85,B 0,C 180,E1 26839.805,E2 26839.805} C_VEL
LIN {X 0,Y 52.098,Z 854.418,A -85,B 0,C 180,E1 26863.403,E2 26863.403} C_VEL
LIN {X 0,Y 42.484,Z 856.971,A -85,B 0,C 180,E1 26889.122,E2 26889.122} C_VEL
LIN {X 0,Y 41.324,Z 857.464,A -85,B 0,C 180,E1 26910,E2 26910} C_VEL
LIN {X 0,Y 48.045,Z 855.563,A -85,B 0,C 180,E1 26949.07,E2 26949.07} C_VEL
LIN {X 0,Y 74.591,Z 847.692,A -85,B 0,C 180,E1 26977.205,E2 26977.205} C_VEL
LIN {X 0,Y 105.72,Z 835.096,A -85,B 0,C 180,E1 26988.817,E2 26988.817} C_VEL
LIN {X 0,Y 140.525,Z 815.324,A -85,B 0,C 180,E1 26995.29,E2 26995.29} C_VEL
LIN {X 0,Y 156.64,Z 803.674,A -85,B 0,C 180,E1 26997.218,E2 26997.218} C_VEL
LIN {X 0,Y 158.438,Z 802.071,A -85,B 0,C 180,E1 26998.405,E2 26998.405} C_VEL
LIN {X 0,Y 158.849,Z 801.57,A -85,B 0,C 180,E1 27000.01,E2 27000.01} C_VEL
LIN {X 0,Y 154.593,Z 805.3,A -85,B 0,C 180,E1 27007.586,E2 27007.586} C_VEL
LIN {X 0,Y 150.59,Z 821.237,A -85,B 0,C 180,E1 27033.583,E2 27033.583} C_VEL
LIN {X 0,Y 162.167,Z 829.87,A -85,B 0,C 180,E1 27049.19,E2 27049.19} C_VEL
LIN {X 0,Y 173.754,Z 837.307,A -85,B 0,C 180,E1 27060.634,E2 27060.634} C_VEL
LIN {X 0,Y 182.042,Z 842.864,A -85,B 0,C 180,E1 27069.078,E2 27069.078} C_VEL
LIN {X 0,Y 187.153,Z 846.893,A -85,B 0,C 180,E1 27076.144,E2 27076.144} C_VEL
LIN {X 0,Y 190.028,Z 848.853,A -85,B 0,C 180,E1 27080.831,E2 27080.831} C_VEL
LIN {X 0,Y 192.389,Z 850.073,A -85,B 0,C 180,E1 27085.486,E2 27085.486} C_VEL
LIN {X 0,Y 193.485,Z 850.429,A -85,B 0,C 180,E1 27090,E2 27090} C_VEL
LIN {X 0,Y 192.409,Z 850.066,A -85,B 0,C 180,E1 27094.513,E2 27094.513} C_VEL
LIN {X 0,Y 190.018,Z 848.854,A -85,B 0,C 180,E1 27099.17,E2 27099.17} C_VEL
LIN {X 0,Y 185.238,Z 845.462,A -85,B 0,C 180,E1 27106.623,E2 27106.623} C_VEL
LIN {X 0,Y 180.47,Z 841.749,A -85,B 0,C 180,E1 27112.637,E2 27112.637} C_VEL
LIN {X 0,Y 173.814,Z 837.266,A -85,B 0,C 180,E1 27119.402,E2 27119.402} C_VEL
LIN {X 0,Y 164.413,Z 831.284,A -85,B 0,C 180,E1 27128.479,E2 27128.479} C_VEL
LIN {X 0,Y 152.102,Z 822.902,A -85,B 0,C 180,E1 27143.316,E2 27143.316} C_VEL
LIN {X 0,Y 154.561,Z 805.319,A -85,B 0,C 180,E1 27172.441,E2 27172.441} C_VEL
LIN {X 0,Y 158.776,Z 801.627,A -85,B 0,C 180,E1 27179.99,E2 27179.99} C_VEL
LIN {X 0,Y 158.308,Z 802.259,A -85,B 0,C 180,E1 27182.169,E2 27182.169} C_VEL
LIN {X 0,Y 151.664,Z 807.464,A -85,B 0,C 180,E1 27183.347,E2 27183.347} C_VEL
LIN {X 0,Y 145.938,Z 811.562,A -85,B 0,C 180,E1 27184.018,E2 27184.018} C_VEL
LIN {X 0,Y 131.139,Z 820.978,A -85,B 0,C 180,E1 27184.285,E2 27184.285} C_VEL
LIN {X 0,Y 115.741,Z 829.313,A -85,B 0,C 180,E1 27184.713,E2 27184.713} C_VEL
LIN {X 0,Y 81.561,Z 844.164,A -85,B 0,C 180,E1 27192.947,E2 27192.947} C_VEL
LIN {X 0,Y 52.396,Z 852.985,A -85,B 0,C 180,E1 27209.9,E2 27209.9} C_VEL
LIN {X 0,Y 35.128,Z 856.735,A -85,B 0,C 180,E1 27244.469,E2 27244.469} C_VEL
LIN {X 0,Y 33.382,Z 857.229,A -85,B 0,C 180,E1 27270,E2 27270} C_VEL
LIN {X 0,Y 42.117,Z 855.325,A -85,B 0,C 180,E1 27315.97,E2 27315.97} C_VEL
LIN {X 0,Y 71.277,Z 847.628,A -85,B 0,C 180,E1 27342.919,E2 27342.919} C_VEL
LIN {X 0,Y 103.12,Z 835.496,A -85,B 0,C 180,E1 27352.9,E2 27352.9} C_VEL
LIN {X 0,Y 138.214,Z 816.264,A -85,B 0,C 180,E1 27358.369,E2 27358.369} C_VEL
LIN {X 0,Y 152.429,Z 806.494,A -85,B 0,C 180,E1 27360.01,E2 27360.01} C_VEL
LIN {X 0,Y 147.518,Z 810.274,A -85,B 0,C 180,E1 27367.729,E2 27367.729} C_VEL
LIN {X 0,Y 145.985,Z 826.893,A -85,B 0,C 180,E1 27398.494,E2 27398.494} C_VEL
LIN {X 0,Y 155.992,Z 833.242,A -85,B 0,C 180,E1 27410.952,E2 27410.952} C_VEL
LIN {X 0,Y 165.793,Z 838.914,A -85,B 0,C 180,E1 27420.794,E2 27420.794} C_VEL
LIN {X 0,Y 174.484,Z 844.19,A -85,B 0,C 180,E1 27429.69,E2 27429.69} C_VEL
LIN {X 0,Y 180.202,Z 848.337,A -85,B 0,C 180,E1 27438.093,E2 27438.093} C_VEL
LIN {X 0,Y 184.232,Z 850.334,A -85,B 0,C 180,E1 27445.286,E2 27445.286} C_VEL
LIN {X 0,Y 185.545,Z 850.758,A -85,B 0,C 180,E1 27450,E2 27450} C_VEL
LIN {X 0,Y 183.039,Z 849.882,A -85,B 0,C 180,E1 27456.918,E2 27456.918} C_VEL
LIN {X 0,Y 178.465,Z 847.061,A -85,B 0,C 180,E1 27464.745,E2 27464.745} C_VEL
LIN {X 0,Y 172.868,Z 843.155,A -85,B 0,C 180,E1 27472.091,E2 27472.091} C_VEL
LIN {X 0,Y 164.062,Z 837.831,A -85,B 0,C 180,E1 27481.034,E2 27481.034} C_VEL
LIN {X 0,Y 153.106,Z 831.572,A -85,B 0,C 180,E1 27492.118,E2 27492.118} C_VEL
LIN {X 0,Y 141.607,Z 818.227,A -85,B 0,C 180,E1 27519.2,E2 27519.2} C_VEL
LIN {X 0,Y 149.113,Z 808.868,A -85,B 0,C 180,E1 27534.505,E2 27534.505} C_VEL
LIN {X 0,Y 152.349,Z 806.55,A -85,B 0,C 180,E1 27539.99,E2 27539.99} C_VEL
LIN {X 0,Y 117.686,Z 828.307,A -85,B 0,C 180,E1 27544.399,E2 27544.399} C_VEL
LIN {X 0,Y 115.741,Z 829.313,A -85,B 0,C 180,E1 27544.713,E2 27544.713} C_VEL
LIN {X 0,Y 99.835,Z 836.6,A -85,B 0,C 180,E1 27545.4,E2 27545.4} C_VEL
LIN {X 0,Y 83.498,Z 842.752,A -85,B 0,C 180,E1 27546.424,E2 27546.424} C_VEL
LIN {X 0,Y 48.871,Z 852.748,A -85,B 0,C 180,E1 27561.656,E2 27561.656} C_VEL
LIN {X 0,Y 28.145,Z 856.499,A -85,B 0,C 180,E1 27597.456,E2 27597.456} C_VEL
LIN {X 0,Y 25.466,Z 856.995,A -85,B 0,C 180,E1 27630,E2 27630} C_VEL
LIN {X 0,Y 36.972,Z 855.086,A -85,B 0,C 180,E1 27684.989,E2 27684.989} C_VEL
LIN {X 0,Y 69.333,Z 847.391,A -85,B 0,C 180,E1 27709.321,E2 27709.321} C_VEL
LIN {X 0,Y 102.306,Z 835.312,A -85,B 0,C 180,E1 27717.376,E2 27717.376} C_VEL
LIN {X 0,Y 138.032,Z 816.145,A -85,B 0,C 180,E1 27721.701,E2 27721.701} C_VEL
LIN {X 0,Y 142.303,Z 813.441,A -85,B 0,C 180,E1 27722.047,E2 27722.047} C_VEL
LIN {X 0,Y 144.029,Z 812.261,A -85,B 0,C 180,E1 27722.765,E2 27722.765} C_VEL
LIN {X 0,Y 137.804,Z 829.263,A -85,B 0,C 180,E1 27757.19,E2 27757.19} C_VEL
LIN {X 0,Y 149.59,Z 836.189,A -85,B 0,C 180,E1 27772.607,E2 27772.607} C_VEL
LIN {X 0,Y 158.316,Z 840.771,A -85,B 0,C 180,E1 27781.434,E2 27781.434} C_VEL
LIN {X 0,Y 167.127,Z 845.498,A -85,B 0,C 180,E1 27790.609,E2 27790.609} C_VEL
LIN {X 0,Y 173.288,Z 849.36,A -85,B 0,C 180,E1 27799.936,E2 27799.936} C_VEL
LIN {X 0,Y 176.078,Z 850.577,A -85,B 0,C 180,E1 27805.067,E2 27805.067} C_VEL
LIN {X 0,Y 177.586,Z 850.994,A -85,B 0,C 180,E1 27810,E2 27810} C_VEL
LIN {X 0,Y 176.088,Z 850.577,A -85,B 0,C 180,E1 27814.932,E2 27814.932} C_VEL
LIN {X 0,Y 171.22,Z 848.236,A -85,B 0,C 180,E1 27823.389,E2 27823.389} C_VEL
LIN {X 0,Y 165.291,Z 844.483,A -85,B 0,C 180,E1 27831.494,E2 27831.494} C_VEL
LIN {X 0,Y 157.132,Z 840.038,A -85,B 0,C 180,E1 27839.849,E2 27839.849} C_VEL
LIN {X 0,Y 147.036,Z 834.887,A -85,B 0,C 180,E1 27850.122,E2 27850.122} C_VEL
LIN {X 0,Y 134.434,Z 824.843,A -85,B 0,C 180,E1 27873.212,E2 27873.212} C_VEL
LIN {X 0,Y 143.966,Z 812.305,A -85,B 0,C 180,E1 27897.233,E2 27897.233} C_VEL
LIN {X 0,Y 139.727,Z 815.1,A -85,B 0,C 180,E1 27898.16,E2 27898.16} C_VEL
LIN {X 0,Y 106.047,Z 833.552,A -85,B 0,C 180,E1 27901.986,E2 27901.986} C_VEL
LIN {X 0,Y 83.498,Z 842.752,A -85,B 0,C 180,E1 27906.424,E2 27906.424} C_VEL
LIN {X 0,Y 66.812,Z 847.813,A -85,B 0,C 180,E1 27908.003,E2 27908.003} C_VEL
LIN {X 0,Y 49.917,Z 851.74,A -85,B 0,C 180,E1 27910.588,E2 27910.588} C_VEL
LIN {X 0,Y 21.825,Z 856.261,A -85,B 0,C 180,E1 27946.074,E2 27946.074} C_VEL
LIN {X 0,Y 17.518,Z 856.76,A -85,B 0,C 180,E1 27990,E2 27990} C_VEL
LIN {X 0,Y 33.022,Z 854.846,A -85,B 0,C 180,E1 28056.493,E2 28056.493} C_VEL
LIN {X 0,Y 68.297,Z 847.154,A -85,B 0,C 180,E1 28076.024,E2 28076.024} C_VEL
LIN {X 0,Y 102.257,Z 835.069,A -85,B 0,C 180,E1 28081.928,E2 28081.928} C_VEL
LIN {X 0,Y 133.504,Z 818.964,A -85,B 0,C 180,E1 28084.718,E2 28084.718} C_VEL
LIN {X 0,Y 135.033,Z 818.066,A -85,B 0,C 180,E1 28085.408,E2 28085.408} C_VEL
LIN {X 0,Y 131.272,Z 832.752,A -85,B 0,C 180,E1 28118.946,E2 28118.946} C_VEL
LIN {X 0,Y 141.309,Z 838.064,A -85,B 0,C 180,E1 28132.301,E2 28132.301} C_VEL
LIN {X 0,Y 152.199,Z 843.112,A -85,B 0,C 180,E1 28143.567,E2 28143.567} C_VEL
LIN {X 0,Y 159.668,Z 846.741,A -85,B 0,C 180,E1 28151.511,E2 28151.511} C_VEL
LIN {X 0,Y 164.854,Z 849.616,A -85,B 0,C 180,E1 28159.416,E2 28159.416} C_VEL
LIN {X 0,Y 167.836,Z 850.823,A -85,B 0,C 180,E1 28164.824,E2 28164.824} C_VEL
LIN {X 0,Y 169.611,Z 851.229,A -85,B 0,C 180,E1 28170,E2 28170} C_VEL
LIN {X 0,Y 167.431,Z 850.704,A -85,B 0,C 180,E1 28175.825,E2 28175.825} C_VEL
LIN {X 0,Y 162.666,Z 848.499,A -85,B 0,C 180,E1 28184.107,E2 28184.107} C_VEL
LIN {X 0,Y 159.663,Z 846.744,A -85,B 0,C 180,E1 28188.484,E2 28188.484} C_VEL
LIN {X 0,Y 152.249,Z 843.081,A -85,B 0,C 180,E1 28196.471,E2 28196.471} C_VEL
LIN {X 0,Y 141.282,Z 838.084,A -85,B 0,C 180,E1 28207.678,E2 28207.678} C_VEL
LIN {X 0,Y 128.171,Z 830.053,A -85,B 0,C 180,E1 28228.325,E2 28228.325} C_VEL
LIN {X 0,Y 135.017,Z 818.075,A -85,B 0,C 180,E1 28254.597,E2 28254.597} C_VEL
LIN {X 0,Y 133.477,Z 818.98,A -85,B 0,C 180,E1 28255.291,E2 28255.291} C_VEL
LIN {X 0,Y 98.447,Z 836.637,A -85,B 0,C 180,E1 28258.499,E2 28258.499} C_VEL
LIN {X 0,Y 60.912,Z 849.226,A -85,B 0,C 180,E1 28266.143,E2 28266.143} C_VEL
LIN {X 0,Y 49.917,Z 851.74,A -85,B 0,C 180,E1 28270.588,E2 28270.588} C_VEL
LIN {X 0,Y 33.042,Z 854.638,A -85,B 0,C 180,E1 28275.588,E2 28275.588} C_VEL
LIN {X 0,Y 16.283,Z 856.052,A -85,B 0,C 180,E1 28288.725,E2 28288.725} C_VEL
LIN {X 0,Y 9.579,Z 856.525,A -85,B 0,C 180,E1 28350.001,E2 28350.001} C_VEL
LIN {X 0,Y 30.709,Z 854.605,A -85,B 0,C 180,E1 28430.424,E2 28430.424} C_VEL
LIN {X 0,Y 68.215,Z 846.917,A -85,B 0,C 180,E1 28442.825,E2 28442.825} C_VEL
LIN {X 0,Y 102.849,Z 834.827,A -85,B 0,C 180,E1 28446.445,E2 28446.445} C_VEL
LIN {X 0,Y 125.594,Z 823.764,A -85,B 0,C 180,E1 28448.057,E2 28448.057} C_VEL
LIN {X 0,Y 127.687,Z 837.451,A -85,B 0,C 180,E1 28485.368,E2 28485.368} C_VEL
LIN {X 0,Y 136.958,Z 841.506,A -85,B 0,C 180,E1 28496.444,E2 28496.444} C_VEL
LIN {X 0,Y 147.622,Z 845.858,A -85,B 0,C 180,E1 28507.401,E2 28507.401} C_VEL
LIN {X 0,Y 152.332,Z 847.873,A -85,B 0,C 180,E1 28512.652,E2 28512.652} C_VEL
LIN {X 0,Y 156.352,Z 849.874,A -85,B 0,C 180,E1 28518.833,E2 28518.833} C_VEL
LIN {X 0,Y 159.604,Z 851.069,A -85,B 0,C 180,E1 28524.557,E2 28524.557} C_VEL
LIN {X 0,Y 161.614,Z 851.466,A -85,B 0,C 180,E1 28530,E2 28530} C_VEL
LIN {X 0,Y 159.604,Z 851.069,A -85,B 0,C 180,E1 28535.443,E2 28535.443} C_VEL
LIN {X 0,Y 155.322,Z 849.406,A -85,B 0,C 180,E1 28542.859,E2 28542.859} C_VEL
LIN {X 0,Y 150.258,Z 847.034,A -85,B 0,C 180,E1 28549.687,E2 28549.687} C_VEL
LIN {X 0,Y 143.107,Z 843.99,A -85,B 0,C 180,E1 28557.247,E2 28557.247} C_VEL
LIN {X 0,Y 133.426,Z 840.016,A -85,B 0,C 180,E1 28567.392,E2 28567.392} C_VEL
LIN {X 0,Y 120.53,Z 832.5,A -85,B 0,C 180,E1 28589.823,E2 28589.823} C_VEL
LIN {X 0,Y 125.58,Z 823.771,A -85,B 0,C 180,E1 28611.947,E2 28611.947} C_VEL
LIN {X 0,Y 91.27,Z 839.45,A -85,B 0,C 180,E1 28614.458,E2 28614.458} C_VEL
LIN {X 0,Y 53.961,Z 850.468,A -85,B 0,C 180,E1 28619.971,E2 28619.971} C_VEL
LIN {X 0,Y 30.707,Z 854.605,A -85,B 0,C 180,E1 28629.556,E2 28629.556} C_VEL
LIN {X 0,Y 16.283,Z 856.052,A -85,B 0,C 180,E1 28648.725,E2 28648.725} C_VEL
LIN {X 0,Y 6.266,Z 856.401,A -85,B 0,C 180,E1 28698.067,E2 28698.067} C_VEL
LIN {X 0,Y 19.976,Z 855.335,A -85,B 0,C 180,E1 28803.252,E2 28803.252} C_VEL
LIN {X 0,Y 54.566,Z 850.233,A -85,B 0,C 180,E1 28808.578,E2 28808.578} C_VEL
LIN {X 0,Y 92.404,Z 839.214,A -85,B 0,C 180,E1 28810.545,E2 28810.545} C_VEL
LIN {X 0,Y 116.108,Z 829.15,A -85,B 0,C 180,E1 28811.53,E2 28811.53} C_VEL
LIN {X 0,Y 121.839,Z 840.414,A -85,B 0,C 180,E1 28848.227,E2 28848.227} C_VEL
LIN {X 0,Y 131.944,Z 844.19,A -85,B 0,C 180,E1 28859.885,E2 28859.885} C_VEL
LIN {X 0,Y 142.985,Z 848.166,A -85,B 0,C 180,E1 28871.478,E2 28871.478} C_VEL
LIN {X 0,Y 147.869,Z 850.133,A -85,B 0,C 180,E1 28878.183,E2 28878.183} C_VEL
LIN {X 0,Y 151.906,Z 851.472,A -85,B 0,C 180,E1 28885.447,E2 28885.447} C_VEL
LIN {X 0,Y 153.592,Z 851.703,A -85,B 0,C 180,E1 28890,E2 28890} C_VEL
LIN {X 0,Y 151.274,Z 851.318,A -85,B 0,C 180,E1 28895.744,E2 28895.744} C_VEL
LIN {X 0,Y 147.859,Z 850.133,A -85,B 0,C 180,E1 28901.818,E2 28901.818} C_VEL
LIN {X 0,Y 143.004,Z 848.165,A -85,B 0,C 180,E1 28908.519,E2 28908.519} C_VEL
LIN {X 0,Y 132.03,Z 844.18,A -85,B 0,C 180,E1 28920.109,E2 28920.109} C_VEL
LIN {X 0,Y 121.738,Z 840.464,A -85,B 0,C 180,E1 28931.72,E2 28931.72} C_VEL
LIN {X 0,Y 116.099,Z 829.154,A -85,B 0,C 180,E1 28968.472,E2 28968.472} C_VEL
LIN {X 0,Y 80.977,Z 843.135,A -85,B 0,C 180,E1 28969.922,E2 28969.922} C_VEL
LIN {X 0,Y 45.844,Z 852.03,A -85,B 0,C 180,E1 28972.219,E2 28972.219} C_VEL
LIN {X 0,Y 13.331,Z 855.875,A -85,B 0,C 180,E1 28980.062,E2 28980.062} C_VEL
LIN {X 0,Y 1.624,Z 856.29,A -85,B 0,C 180,E1 29070.005,E2 29070.005} C_VEL
LIN {X 0,Y 19.976,Z 855.335,A -85,B 0,C 180,E1 29163.252,E2 29163.252} C_VEL
LIN {X 0,Y 32.629,Z 854.041,A -85,B 0,C 180,E1 29170.535,E2 29170.535} C_VEL
LIN {X 0,Y 51.717,Z 850.958,A -85,B 0,C 180,E1 29176.988,E2 29176.988} C_VEL
LIN {X 0,Y 53.876,Z 850.509,A -85,B 0,C 180,E1 29176.925,E2 29176.925} C_VEL
LIN {X 0,Y 90.549,Z 840.349,A -85,B 0,C 180,E1 29175.473,E2 29175.473} C_VEL
LIN {X 0,Y 107.063,Z 833.905,A -85,B 0,C 180,E1 29175.543,E2 29175.543} C_VEL
LIN {X 0,Y 116.179,Z 843.186,A -85,B 0,C 180,E1 29211.456,E2 29211.456} C_VEL
LIN {X 0,Y 127.41,Z 846.691,A -85,B 0,C 180,E1 29223.978,E2 29223.978} C_VEL
LIN {X 0,Y 133.384,Z 848.47,A -85,B 0,C 180,E1 29230.091,E2 29230.091} C_VEL
LIN {X 0,Y 139.361,Z 850.529,A -85,B 0,C 180,E1 29237.943,E2 29237.943} C_VEL
LIN {X 0,Y 142.881,Z 851.569,A -85,B 0,C 180,E1 29243.917,E2 29243.917} C_VEL
LIN {X 0,Y 145.571,Z 851.94,A -85,B 0,C 180,E1 29250,E2 29250} C_VEL
LIN {X 0,Y 142.877,Z 851.569,A -85,B 0,C 180,E1 29256.083,E2 29256.083} C_VEL
LIN {X 0,Y 138.949,Z 850.405,A -85,B 0,C 180,E1 29262.587,E2 29262.587} C_VEL
LIN {X 0,Y 133.464,Z 848.467,A -85,B 0,C 180,E1 29269.897,E2 29269.897} C_VEL
LIN {X 0,Y 123.114,Z 845.387,A -85,B 0,C 180,E1 29280.566,E2 29280.566} C_VEL
LIN {X 0,Y 110.434,Z 841.116,A -85,B 0,C 180,E1 29296.708,E2 29296.708} C_VEL
LIN {X 0,Y 106.987,Z 833.94,A -85,B 0,C 180,E1 29324.439,E2 29324.439} C_VEL
LIN {X 0,Y 70.876,Z 846.444,A -85,B 0,C 180,E1 29324.007,E2 29324.007} C_VEL
LIN {X 0,Y 32.231,Z 854.123,A -85,B 0,C 180,E1 29319.965,E2 29319.965} C_VEL
LIN {X 0,Y 6.319,Z 856.055,A -85,B 0,C 180,E1 29249.999,E2 29249.999} C_VEL
LIN {X 0,Y 32.227,Z 854.123,A -85,B 0,C 180,E1 29180.011,E2 29180.011} C_VEL
LIN {X 0,Y 53.876,Z 850.509,A -85,B 0,C 180,E1 29176.925,E2 29176.925} C_VEL
LIN {X 0,Y 70.812,Z 846.692,A -85,B 0,C 180,E1 29179.231,E2 29179.231} C_VEL
LIN {X 0,Y 87.574,Z 841.92,A -85,B 0,C 180,E1 29180.705,E2 29180.705} C_VEL
LIN {X 0,Y 96.679,Z 838.741,A -85,B 0,C 180,E1 29180.008,E2 29180.008} C_VEL
LIN {X 0,Y 98.193,Z 838.616,A -85,B 0,C 180,E1 29182.308,E2 29182.308} C_VEL
LIN {X 0,Y 110.785,Z 845.625,A -85,B 0,C 180,E1 29215.106,E2 29215.106} C_VEL
LIN {X 0,Y 118.436,Z 847.615,A -85,B 0,C 180,E1 29223.515,E2 29223.515} C_VEL
LIN {X 0,Y 126.884,Z 849.864,A -85,B 0,C 180,E1 29232.705,E2 29232.705} C_VEL
LIN {X 0,Y 129.737,Z 850.687,A -85,B 0,C 180,E1 29236.502,E2 29236.502} C_VEL
LIN {X 0,Y 134.403,Z 851.822,A -85,B 0,C 180,E1 29243.532,E2 29243.532} C_VEL
LIN {X 0,Y 137.469,Z 852.179,A -85,B 0,C 180,E1 29250,E2 29250} C_VEL
LIN {X 0,Y 134.402,Z 851.822,A -85,B 0,C 180,E1 29256.468,E2 29256.468} C_VEL
LIN {X 0,Y 129.758,Z 850.687,A -85,B 0,C 180,E1 29263.495,E2 29263.495} C_VEL
LIN {X 0,Y 122.978,Z 848.802,A -85,B 0,C 180,E1 29271.675,E2 29271.675} C_VEL
LIN {X 0,Y 112.975,Z 846.223,A -85,B 0,C 180,E1 29282.416,E2 29282.416} C_VEL
LIN {X 0,Y 99.909,Z 841.87,A -85,B 0,C 180,E1 29302.669,E2 29302.669} C_VEL
LIN {X 0,Y 98.102,Z 838.623,A -85,B 0,C 180,E1 29317.821,E2 29317.821} C_VEL
LIN {X 0,Y 96.697,Z 838.739,A -85,B 0,C 180,E1 29319.961,E2 29319.961} C_VEL
LIN {X 0,Y 60.192,Z 849.549,A -85,B 0,C 180,E1 29315.914,E2 29315.914} C_VEL
LIN {X 0,Y 35.81,Z 853.882,A -85,B 0,C 180,E1 29307.737,E2 29307.737} C_VEL
LIN {X 0,Y 14.283,Z 855.82,A -85,B 0,C 180,E1 29249.999,E2 29249.999} C_VEL
LIN {X 0,Y 35.802,Z 853.882,A -85,B 0,C 180,E1 29192.244,E2 29192.244} C_VEL
LIN {X 0,Y 73.546,Z 846.205,A -85,B 0,C 180,E1 29182.121,E2 29182.121} C_VEL
LIN {X 0,Y 87.574,Z 841.92,A -85,B 0,C 180,E1 29180.705,E2 29180.705} C_VEL
LIN {X 0,Y 90.663,Z 841.227,A -85,B 0,C 180,E1 29182.586,E2 29182.586} C_VEL
LIN {X 0,Y 91.494,Z 842.056,A -85,B 0,C 180,E1 29188.431,E2 29188.431} C_VEL
LIN {X 0,Y 91.801,Z 843.61,A -85,B 0,C 180,E1 29195.605,E2 29195.605} C_VEL
LIN {X 0,Y 105.859,Z 847.748,A -85,B 0,C 180,E1 29219.135,E2 29219.135} C_VEL
LIN {X 0,Y 114.153,Z 849.579,A -85,B 0,C 180,E1 29228.223,E2 29228.223} C_VEL
LIN {X 0,Y 120.556,Z 850.97,A -85,B 0,C 180,E1 29235.453,E2 29235.453} C_VEL
LIN {X 0,Y 125.691,Z 852.083,A -85,B 0,C 180,E1 29243.081,E2 29243.081} C_VEL
LIN {X 0,Y 129.403,Z 852.418,A -85,B 0,C 180,E1 29250,E2 29250} C_VEL
LIN {X 0,Y 125.695,Z 852.083,A -85,B 0,C 180,E1 29256.918,E2 29256.918} C_VEL
LIN {X 0,Y 120.599,Z 850.968,A -85,B 0,C 180,E1 29264.542,E2 29264.542} C_VEL
LIN {X 0,Y 112.159,Z 849.152,A -85,B 0,C 180,E1 29273.89,E2 29273.89} C_VEL
LIN {X 0,Y 105.838,Z 847.757,A -85,B 0,C 180,E1 29280.846,E2 29280.846} C_VEL
LIN {X 0,Y 90.377,Z 841.916,A -85,B 0,C 180,E1 29313.878,E2 29313.878} C_VEL
LIN {X 0,Y 69.437,Z 848.039,A -85,B 0,C 180,E1 29310.713,E2 29310.713} C_VEL
LIN {X 0,Y 40.695,Z 853.641,A -85,B 0,C 180,E1 29298.082,E2 29298.082} C_VEL
LIN {X 0,Y 22.228,Z 855.585,A -85,B 0,C 180,E1 29250,E2 29250} C_VEL
LIN {X 0,Y 40.686,Z 853.641,A -85,B 0,C 180,E1 29201.904,E2 29201.904} C_VEL
LIN {X 0,Y 76.963,Z 845.968,A -85,B 0,C 180,E1 29187.717,E2 29187.717} C_VEL
LIN {X 0,Y 88.017,Z 842.603,A -85,B 0,C 180,E1 29185.882,E2 29185.882} C_VEL
LIN {X 0,Y 90.519,Z 841.888,A -85,B 0,C 180,E1 29186.202,E2 29186.202} C_VEL
LIN {X 0,Y 91.801,Z 843.61,A -85,B 0,C 180,E1 29195.605,E2 29195.605} C_VEL
LIN {X 0,Y 92.231,Z 846.261,A -85,B 0,C 180,E1 29206.373,E2 29206.373} C_VEL
LIN {X 0,Y 95.01,Z 848.569,A -85,B 0,C 180,E1 29216.951,E2 29216.951} C_VEL
LIN {X 0,Y 101.198,Z 849.653,A -85,B 0,C 180,E1 29223.885,E2 29223.885} C_VEL
LIN {X 0,Y 110.47,Z 851.282,A -85,B 0,C 180,E1 29234.091,E2 29234.091} C_VEL
LIN {X 0,Y 117.009,Z 852.344,A -85,B 0,C 180,E1 29242.565,E2 29242.565} C_VEL
LIN {X 0,Y 121.147,Z 852.662,A -85,B 0,C 180,E1 29250.037,E2 29250.037} C_VEL
LIN {X 0,Y 117.017,Z 852.343,A -85,B 0,C 180,E1 29257.434,E2 29257.434} C_VEL
LIN {X 0,Y 110.319,Z 851.256,A -85,B 0,C 180,E1 29266.073,E2 29266.073} C_VEL
LIN {X 0,Y 100.508,Z 849.537,A -85,B 0,C 180,E1 29276.867,E2 29276.867} C_VEL
LIN {X 0,Y 86.949,Z 846.781,A -85,B 0,C 180,E1 29295.828,E2 29295.828} C_VEL
LIN {X 0,Y 83.432,Z 845.193,A -85,B 0,C 180,E1 29306.994,E2 29306.994} C_VEL
LIN {X 0,Y 66.567,Z 849.494,A -85,B 0,C 180,E1 29302.756,E2 29302.756} C_VEL
LIN {X 0,Y 35.762,Z 854.831,A -85,B 0,C 180,E1 29275.047,E2 29275.047} C_VEL
LIN {X 0,Y 30.317,Z 855.337,A -85,B 0,C 180,E1 29248.554,E2 29248.554} C_VEL
LIN {X 0,Y 51.977,Z 852.449,A -85,B 0,C 180,E1 29204.816,E2 29204.816} C_VEL
LIN {X 0,Y 78.332,Z 846.5,A -85,B 0,C 180,E1 29193.5,E2 29193.5} C_VEL
LIN {X 0,Y 83.525,Z 845.163,A -85,B 0,C 180,E1 29192.964,E2 29192.964} C_VEL
LIN {X 0,Y 95.01,Z 848.569,A -85,B 0,C 180,E1 29216.951,E2 29216.951} C_VEL
LIN {X 0,Y 98.266,Z 850.095,A -85,B 0,C 180,E1 29224.444,E2 29224.444} C_VEL
LIN {X 0,Y 103.001,Z 852.093,A -85,B 0,C 180,E1 29236.946,E2 29236.946} C_VEL
LIN {X 0,Y 107.715,Z 852.622,A -85,B 0,C 180,E1 29241.92,E2 29241.92} C_VEL
